ACTION removeLens_active:
IF removeLens._x AND removeLens.x = FALSE THEN
	timer.IN := FALSE;
	timer2.IN := FALSE;
	trn_removeLensDone := FALSE;
	var_process := 0;
ELSIF removeLens._x AND removeLens.x THEN
	CASE var_process OF
		0://insert parameter
			fbi_gm_removeLens.p_Init := TRUE;
			gvl_axis.fbi_motionControler.in_var_targetPosX := gvl_param.var_productInfo[gvl_param.var_currentProductID].teachPos.remove.x;
			gvl_axis.fbi_motionControler.in_var_targetPosY := gvl_param.var_productInfo[gvl_param.var_currentProductID].teachPos.remove.y;
			gvl_axis.fbi_motionControler.in_var_targetPosZ := gvl_param.var_productInfo[gvl_param.var_currentProductID].teachPos.remove.z;
			gvl_axis.fbi_motionControler.in_var_direction := eP_motionDirection.XYZ;
			IF gvl_solv.ref_ejector.input.in_flg_sensVac THEN
				var_process := 1;
			ELSE
				gvl_solv.fbi_ejector.in_var_vacMode := eP_ejeVacMode.break;
				gvl_solv.fbi_ejector.in_flg_run := TRUE;
				var_process := 20;
			END_IF
		1://move start
			gvl_axis.fbi_motionControler.in_flg_start := TRUE;
			IF gvl_axis.fbi_motionControler.out_flg_Done THEN
				var_process := 2;
			END_IF
		2://insert ejector parameter
			gvl_axis.fbi_motionControler.in_flg_start := FALSE;
			gvl_solv.fbi_ejector.in_flg_run := FALSE;
			gvl_solv.fbi_ejector.in_var_vacMode := eP_ejeVacMode.break;
			var_process := 3;
		3://break
			gvl_solv.fbi_ejector.in_flg_run := TRUE;
			IF gvl_solv.fbi_ejector.out_flg_Done THEN
				gvl_solv.fbi_ejector.in_flg_run := FALSE;
				var_process := 4;
			END_IF
		4://insert initial position
			gvl_solv.fbi_ejector.in_flg_run := FALSE;
			gvl_solv.fbi_chuck.in_var_moveMode := eP_svMoveMode.svA;
			gvl_axis.fbi_motionControler.in_var_targetPosX := gvl_param.var_productInfo[gvl_param.var_currentProductID].teachPos.initial.x;
			gvl_axis.fbi_motionControler.in_var_targetPosY := gvl_param.var_productInfo[gvl_param.var_currentProductID].teachPos.initial.y;
			gvl_axis.fbi_motionControler.in_var_targetPosZ := gvl_param.var_productInfo[gvl_param.var_currentProductID].teachPos.initial.z;
			gvl_axis.fbi_motionControler.in_var_direction := eP_motionDirection.ZYX;
			var_process := 5;
		5://move to initial position
			gvl_axis.fbi_motionControler.in_flg_start := TRUE;
			IF gvl_axis.fbi_motionControler.out_flg_Done THEN
				gvl_solv.fbi_gm_push.in_flg_run := FALSE;
				gvl_solv.fbi_gm_chuck.in_flg_run := FALSE;
				IF gvl_io.flg_fiberSens THEN
					var_process := 6;
				ELSE
					var_process := 20;
				END_IF
			END_IF
		6:
			gvl_solv.fbi_chuck.in_var_moveMode := eP_svMoveMode.svB;
			gvl_solv.fbi_push.in_var_moveMode := eP_svMoveMode.svB;
			gvl_elecylinder.fbi_axisTransport.in_var_moveMode := eP_eleMoveMode.eleB;
			gvl_solv.fbi_ejector.in_var_vacMode := eP_ejeVacMode.halt;
			gvl_axis.fbi_motionControler.in_var_targetPosX := gvl_param.var_productInfo[gvl_param.var_currentProductID].teachPos.pickUp.x;
			gvl_axis.fbi_motionControler.in_var_targetPosY := gvl_param.var_productInfo[gvl_param.var_currentProductID].teachPos.pickUp.y;
			gvl_axis.fbi_motionControler.in_var_targetPosZ := gvl_param.var_productInfo[gvl_param.var_currentProductID].teachPos.pickUp.z;
			gvl_axis.fbi_motionControler.in_var_direction := eP_motionDirection.XYZ;
			var_process := 7;
		7:
			gvl_elecylinder.fbi_axisTransport.in_flg_run := TRUE;
			gvl_solv.fbi_ejector.in_flg_run := TRUE;
			gvl_solv.fbi_chuck.in_flg_run := TRUE;
			gvl_solv.fbi_push.in_flg_run := TRUE;
			var_process := 8;
		8:
			IF gvl_io.in_wire_svChuckClose AND gvl_io.in_wire_svPushClose AND gvl_io.in_flg_eleTransportMoving THEN
				gvl_axis.fbi_motionControler.in_flg_start := TRUE;
				gvl_solv.fbi_ejector.in_flg_run := FALSE;
				gvl_elecylinder.fbi_axisTransport.in_flg_run := FALSE;
				gvl_solv.fbi_chuck.in_flg_run := FALSE;
				gvl_solv.fbi_push.in_flg_run := FALSE;
				var_process := 9;
			END_IF
		9:
			IF gvl_axis.fbi_motionControler.out_flg_Done THEN
				gvl_axis.fbi_motionControler.in_flg_start := FALSE;
				gvl_axis.fbi_motionControler.in_var_targetPosX := gvl_param.var_productInfo[gvl_param.var_currentProductID].teachPos.initial.x;
				gvl_axis.fbi_motionControler.in_var_targetPosY := gvl_param.var_productInfo[gvl_param.var_currentProductID].teachPos.initial.y;
				gvl_axis.fbi_motionControler.in_var_targetPosZ := gvl_param.var_productInfo[gvl_param.var_currentProductID].teachPos.initial.z;
				gvl_axis.fbi_motionControler.in_var_direction := eP_motionDirection.ZYX;
				var_process := 10;
			END_IF
		10:
			gvl_axis.fbi_motionControler.in_flg_start := TRUE;
			var_process := 11;
		11:
			IF gvl_axis.fbi_motionControler.out_flg_Done THEN
				gvl_axis.fbi_motionControler.in_flg_start := FALSE;
				gvl_axis.fbi_motionControler.in_var_targetPosX := gvl_param.var_productInfo[gvl_param.var_currentProductID].teachPos.remove.x;
				gvl_axis.fbi_motionControler.in_var_targetPosY := gvl_param.var_productInfo[gvl_param.var_currentProductID].teachPos.remove.y;
				gvl_axis.fbi_motionControler.in_var_targetPosZ := gvl_param.var_productInfo[gvl_param.var_currentProductID].teachPos.remove.z;
				gvl_axis.fbi_motionControler.in_var_direction := eP_motionDirection.XYZ;
				var_process := 12;
			END_IF
		12:
			gvl_axis.fbi_motionControler.in_flg_start := TRUE;
			gvl_solv.fbi_ejector.in_var_vacMode := eP_ejeVacMode.break;
			var_process := 13;
		13:
			IF gvl_axis.fbi_motionControler.out_flg_Done THEN
				gvl_solv.fbi_ejector.in_flg_run := TRUE;
				var_process := 14;	
			END_IF
		14:
			IF gvl_solv.fbi_ejector.out_flg_Done THEN
				gvl_solv.fbi_ejector.in_flg_run := FALSE;
				gvl_axis.fbi_motionControler.in_var_targetPosX := gvl_param.var_productInfo[gvl_param.var_currentProductID].teachPos.initial.x;
				gvl_axis.fbi_motionControler.in_var_targetPosY := gvl_param.var_productInfo[gvl_param.var_currentProductID].teachPos.initial.y;
				gvl_axis.fbi_motionControler.in_var_targetPosZ := gvl_param.var_productInfo[gvl_param.var_currentProductID].teachPos.initial.z;
				gvl_axis.fbi_motionControler.in_var_direction := eP_motionDirection.ZYX;
				var_process := 15;	
			END_IF
		15:
			gvl_axis.fbi_motionControler.in_flg_start := TRUE;
			gvl_solv.fbi_chuck.in_var_moveMode := eP_svMoveMode.svB;
			gvl_solv.fbi_push.in_var_moveMode := eP_svMoveMode.svB;
			gvl_elecylinder.fbi_axisTransport.in_var_moveMode := eP_eleMoveMode.eleB;
			var_process := 16;
		16:
			IF gvl_axis.fbi_motionControler.out_flg_Done THEN
				IF gvl_axis.fbi_motionControler.out_flg_Done THEN
					gvl_elecylinder.fbi_axisTransport.in_flg_run := TRUE;
					gvl_solv.fbi_chuck.in_flg_run := TRUE;
					gvl_solv.fbi_push.in_flg_run := TRUE;
					var_process := 17;
				END_IF
			END_IF
		17:
			IF gvl_io.in_wire_svChuckOpen AND gvl_io.in_wire_svPushOpen AND gvl_io.in_flg_eleTransportOrigin THEN
				gvl_elecylinder.fbi_axisTransport.in_flg_run := FALSE;
				gvl_solv.fbi_chuck.in_flg_run := FALSE;
				gvl_solv.fbi_push.in_flg_run := FALSE;
				var_process := 20;
			END_IF
		20:
			IF NOT gvl_visu.flg_btn_usingMeasurementSystem THEN
				var_process := 50;
			ELSE
				fbi_gm_removeLens.p_Init := TRUE;
				fbi_gm_removeLens.in_flg_run := FALSE;
				var_process := 21;
			END_IF
		21:
			fbi_gm_removeLens.p_Init := FALSE;
			fbi_gm_removeLens.in_flg_run := TRUE;
			var_process := 22;
		22:
			fbi_gm_removeLens.in_flg_run := FALSE;
			IF fbi_gm_removeLens.out_flg_Done THEN
				var_process := 50;
			END_IF
			
		50:
			gvl_solv.fbi_ejector.in_flg_run := FALSE;
			trn_removeLensDone := TRUE;
	END_CASE
	fbi_gm_removeLens(in_flg_run:= , out_flg_Done=> );
	timer(IN:= , PT:= T#0.5S , Q=> , ET=> );
	timer2(IN:= , PT:= T#0.5S , Q=> , ET=> );
END_IF
END_ACTION

END_FUNCTION_BLOCK

// ---- FBs/fb_lensTranport.TcPOU
FUNCTION_BLOCK fb_lensTranport
VAR_INPUT
END_VAR
VAR_OUTPUT
END_VAR
VAR
	SFCInit: bool;
	trn_wattingForLensDone: BOOL;
	trn_connectionCheckDone: BOOL;
	flg_buf_gateLengthISSuccessed: BOOL;
	flg_buf_dummySignal: BOOL;
	trn_chuckDone: BOOL;
	var_chuckCount: INT;
	trn_transportDone: BOOL;
	trn_waitTakingLensDone: BOOL;
	trn_moveToHomeDone: BOOL;
	fbi_getCav: fb_getCav;
	trn_readCavDone: BOOL;
	trn_gm_chuckDone: BOOL;
	trn_gm_transportDone: BOOL;
	trn_gm_moveToHomeDone: BOOL;
	trn_cavCheckDone: BOOL;
	fbi_delayTimer: TON;
	trn_AddCountDone: BOOL;
	var_process: INT;
	flg_chuckDone: BOOL;
	flg_pushDone: BOOL;
	trn_LensCheckDone: BOOL;
END_VAR

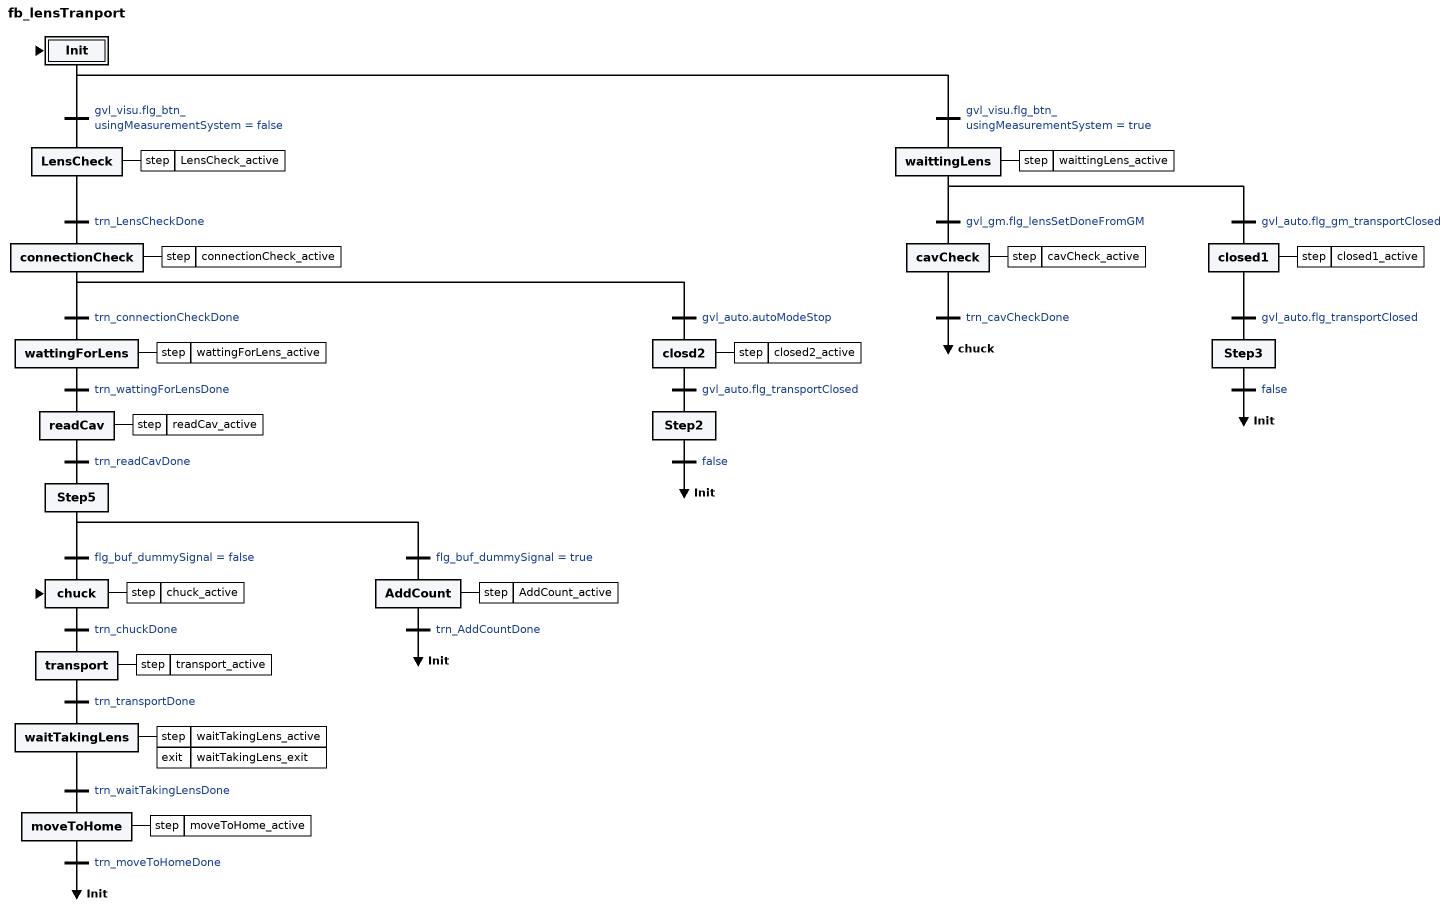
INITIAL_STEP Init:
END_STEP
TRANSITION FROM Init TO LensCheck
    := gvl_visu.flg_btn_usingMeasurementSystem = false;
END_TRANSITION
TRANSITION FROM Init TO waittingLens
    := gvl_visu.flg_btn_usingMeasurementSystem = true;
END_TRANSITION
STEP waittingLens:
    waittingLens_active(N);  // step action
END_STEP
TRANSITION FROM waittingLens TO cavCheck
    := gvl_gm.flg_lensSetDoneFromGM;
END_TRANSITION
STEP cavCheck:
    cavCheck_active(N);  // step action
END_STEP
TRANSITION FROM cavCheck TO chuck
    := trn_cavCheckDone;
END_TRANSITION
TRANSITION FROM waittingLens TO closed1
    := gvl_auto.flg_gm_transportClosed;
END_TRANSITION
STEP closed1:
    closed1_active(N);  // step action
END_STEP
TRANSITION FROM closed1 TO Step3
    := gvl_auto.flg_transportClosed;
END_TRANSITION
STEP Step3:
END_STEP
TRANSITION FROM Step3 TO Init
    := false;
END_TRANSITION
STEP LensCheck:
    LensCheck_active(N);  // step action
END_STEP
TRANSITION FROM LensCheck TO connectionCheck
    := trn_LensCheckDone;
END_TRANSITION
STEP connectionCheck:
    connectionCheck_active(N);  // step action
END_STEP
TRANSITION FROM connectionCheck TO wattingForLens
    := trn_connectionCheckDone;
END_TRANSITION
STEP wattingForLens:
    wattingForLens_active(N);  // step action
END_STEP
TRANSITION FROM wattingForLens TO readCav
    := trn_wattingForLensDone;
END_TRANSITION
TRANSITION FROM connectionCheck TO closd2
    := gvl_auto.autoModeStop;
END_TRANSITION
STEP closd2:
    closed2_active(N);  // step action
END_STEP
TRANSITION FROM closd2 TO Step2
    := gvl_auto.flg_transportClosed;
END_TRANSITION
STEP Step2:
END_STEP
TRANSITION FROM Step2 TO Init
    := false;
END_TRANSITION
STEP readCav:
    readCav_active(N);  // step action
END_STEP
TRANSITION FROM readCav TO Step5
    := trn_readCavDone;
END_TRANSITION
STEP Step5:
END_STEP
TRANSITION FROM Step5 TO chuck
    := flg_buf_dummySignal = false;
END_TRANSITION
TRANSITION FROM Step5 TO AddCount
    := flg_buf_dummySignal = true;
END_TRANSITION
STEP AddCount:
    AddCount_active(N);  // step action
END_STEP
TRANSITION FROM AddCount TO Init
    := trn_AddCountDone;
END_TRANSITION
STEP chuck:
    chuck_active(N);  // step action
END_STEP
TRANSITION FROM chuck TO transport
    := trn_chuckDone;
END_TRANSITION
STEP transport:
    transport_active(N);  // step action
END_STEP
TRANSITION FROM transport TO waitTakingLens
    := trn_transportDone;
END_TRANSITION
STEP waitTakingLens:
    waitTakingLens_active(N);  // step action
    waitTakingLens_exit(P0);  // exit action
END_STEP
TRANSITION FROM waitTakingLens TO moveToHome
    := trn_waitTakingLensDone;
END_TRANSITION
STEP moveToHome:
    moveToHome_active(N);  // step action
END_STEP
TRANSITION FROM moveToHome TO Init
    := trn_moveToHomeDone;
END_TRANSITION

ACTION AddCount_active:
IF AddCount._x AND AddCount.x = FALSE THEN
	trn_AddCountDone := FALSE;
ELSIF AddCount._x AND AddCount.x THEN
	trn_AddCountDone := TRUE;
END_IF
END_ACTION

ACTION cavCheck_active:
IF cavCheck._x AND cavCheck.x = FALSE THEN
	trn_cavCheckDone := FALSE;
ELSIF cavCheck._x AND cavCheck.x THEN
	gvl_auto.cavNo := gvl_gm.var_buf_tranportCav;
	gvl_auto.flg_buf_gateLengthIsPassed := gvl_gm.flg_buf_gateLengthIsPassed;
	trn_cavCheckDone := TRUE;
END_IF
END_ACTION

ACTION chuck_active:
IF chuck._x AND chuck.x = FALSE THEN
	gvl_gm.flg_lensRequest := FALSE;
	trn_chuckDone := FALSE;
	gvl_auto.flg_gateData_Tx := FALSE;
	gvl_solv.fbi_chuck.in_flg_run := FALSE;
	gvl_solv.fbi_push.in_flg_run := FALSE;
	var_chuckCount := -11;
ELSIF chuck._x AND chuck.x THEN
	CASE var_chuckCount OF
		-11:
			IF gvl_param.var_productInfo[gvl_param.var_currentProductID].flg_mode_stocker THEN
				var_chuckCount := -10; // Mode 1
			ELSE
				var_chuckCount := 0;  // Mode 0
			END_IF
		
		// Mode 1: 押す →　解除　→ チャック →　押す
		-10:
			gvl_solv.fbi_push.in_var_moveMode := eP_svMoveMode.svB;
			gvl_solv.fbi_push.in_flg_run := TRUE;
			var_chuckCount := -9;
		-9://close
			IF gvl_solv.fbi_push.out_flg_Done THEN
				gvl_solv.fbi_push.in_flg_run := FALSE;
				var_chuckCount := -8;
			END_IF
		-8:		
			gvl_solv.fbi_push.in_var_moveMode := eP_svMoveMode.svA;
			gvl_solv.fbi_push.in_flg_run := TRUE;
			var_chuckCount := -7;
		-7://open
			IF gvl_solv.fbi_push.out_flg_Done THEN
				gvl_solv.fbi_push.in_flg_run := FALSE;
				var_chuckCount := -6;
			END_IF
		-6:
			gvl_solv.fbi_chuck.in_var_moveMode := eP_svMoveMode.svB;
			gvl_solv.fbi_chuck.in_flg_run := TRUE;
			var_chuckCount := -5;
		-5://push close
			IF gvl_solv.fbi_chuck.out_flg_Done THEN
				gvl_solv.fbi_chuck.in_flg_run := FALSE;
				var_chuckCount := -4;
			END_IF
		-4:
			gvl_solv.fbi_push.in_var_moveMode := eP_svMoveMode.svB;
			gvl_solv.fbi_push.in_flg_run := TRUE;
			var_chuckCount := -3;
		-3://close
			
			IF gvl_solv.fbi_push.out_flg_Done THEN
				gvl_solv.fbi_push.in_flg_run := FALSE;
				var_chuckCount := 12;
			END_IF
		
		// Mode 0: チャック → 解除 → 押す → チャック
		0:
			gvl_solv.fbi_chuck.in_var_moveMode := eP_svMoveMode.svB;
			gvl_solv.fbi_chuck.in_flg_run := TRUE;
			var_chuckCount := 1;
		1://close
			
			IF gvl_solv.fbi_chuck.out_flg_Done THEN
				gvl_solv.fbi_chuck.in_flg_run := FALSE;
				var_chuckCount := 2;
			END_IF
		2:		
			gvl_solv.fbi_chuck.in_var_moveMode := eP_svMoveMode.svA;
			gvl_solv.fbi_chuck.in_flg_run := TRUE;
			var_chuckCount := 3;
		3://open
			
			IF gvl_solv.fbi_chuck.out_flg_Done THEN
				var_chuckCount := 4;
			END_IF
		4:
			gvl_solv.fbi_push.in_var_moveMode := eP_svMoveMode.svB;
			gvl_solv.fbi_push.in_flg_run := TRUE;
			var_chuckCount := 5;
		5://push close
			
			IF gvl_solv.fbi_push.out_flg_Done THEN
				gvl_solv.fbi_push.in_flg_run := FALSE;
				gvl_solv.fbi_chuck.in_flg_run := FALSE;
				var_chuckCount := 6;
			END_IF
		6:
			
			gvl_solv.fbi_chuck.in_var_moveMode := eP_svMoveMode.svB;
			gvl_solv.fbi_chuck.in_flg_run := TRUE;
			var_chuckCount := 7;
		7://close
			
			IF gvl_solv.fbi_chuck.out_flg_Done THEN
				gvl_solv.fbi_chuck.in_flg_run := FALSE;
				var_chuckCount := 12;
			END_IF
		8:
			
			gvl_solv.fbi_chuck.in_var_moveMode := eP_svMoveMode.svA;
			gvl_solv.fbi_chuck.in_flg_run := TRUE;
			var_chuckCount := 9;
		9://open
			
			IF gvl_solv.fbi_chuck.out_flg_Done THEN
				gvl_solv.fbi_chuck.in_flg_run := FALSE;
				var_chuckCount := 10;
			END_IF
		10:
			
			gvl_solv.fbi_chuck.in_var_moveMode := eP_svMoveMode.svB;
			gvl_solv.fbi_chuck.in_flg_run := TRUE;
			var_chuckCount := 11;
		11://close
			
			IF gvl_solv.fbi_chuck.out_flg_Done THEN
				var_chuckCount := 12;
			END_IF
		12://gate measurement
			IF gvl_visu.flg_btn_gateMeasurementIsNone THEN
				IF flg_buf_gateLengthISSuccessed THEN
					gvl_auto.gateLengthIsPassed := TRUE;
				ELSIF gvl_auto.flg_buf_gateLengthIsPassed THEN
					gvl_auto.gateLengthIsPassed := TRUE;
				ELSE
					gvl_auto.gateLengthIsPassed := FALSE;
				END_IF
			ELSE
				IF gvl_io.var_gateLength > gvl_param.var_productInfo[gvl_param.var_currentProductID].gateLength_max OR gvl_io.var_gateLength < gvl_param.var_productInfo[gvl_param.var_currentProductID].gateLength_min THEN
					gvl_auto.gateLengthIsPassed := FALSE;
				ELSE
					gvl_auto.gateLengthIsPassed := TRUE;
				END_IF
				gvl_auto.flg_gateData_Tx := TRUE;
				
			END_IF
			var_chuckCount := 13;
		13:
			gvl_solv.fbi_chuck.in_flg_run := FALSE;
			gvl_elecylinder.fbi_axisRotary.in_flg_run := FALSE;
			gvl_elecylinder.fbi_axisRotary.in_var_moveMode := eP_eleMoveMode.eleB;
			IF gvl_visu.flg_btn_RotaryIsNotUse THEN
				var_chuckCount := 16;
			ELSE
				var_chuckCount := 14;
			END_IF
		14:
			gvl_elecylinder.fbi_axisRotary.in_flg_run := TRUE;
			var_chuckCount := 15;
		15:
			IF gvl_elecylinder.fbi_axisRotary.out_flg_Done THEN
				gvl_elecylinder.fbi_axisRotary.in_flg_run := FALSE;
				var_chuckCount := 16;
			END_IF
		16:
			trn_chuckDone := TRUE;
	END_CASE
END_IF
END_ACTION

ACTION closed1_active:
IF closed1._x AND closed1.x = FALSE THEN
	gvl_auto.flg_transportClosed := FALSE;
	gvl_elecylinder.fbi_axisTransport.in_flg_run := FALSE;
	gvl_elecylinder.fbi_axisRotary.in_flg_run:= FALSE;
	gvl_elecylinder.fbi_axisTransport.in_var_moveMode := eP_eleMoveMode.eleB;
	gvl_elecylinder.fbi_axisRotary.in_var_moveMode:= eP_eleMoveMode.eleB;
	var_process := 0;
ELSIF closed1._x AND closed1.x THEN
	CASE var_process OF
		0:
			gvl_elecylinder.fbi_axisRotary.in_flg_run:= TRUE;
			var_process := 1;
		1:
			IF gvl_elecylinder.fbi_axisRotary.out_flg_Done THEN
				gvl_elecylinder.fbi_axisRotary.in_flg_run:= FALSE;
				var_process := 2;
			END_IF
		2:
			gvl_elecylinder.fbi_axisTransport.in_flg_run := TRUE;
			var_process := 3;
		3:
			IF gvl_elecylinder.fbi_axisTransport.out_flg_Done THEN
				gvl_elecylinder.fbi_axisTransport.in_flg_run:= FALSE;
				gvl_auto.flg_transportClosed := TRUE;
			END_IF
	END_CASE
END_IF
END_ACTION

ACTION closed2_active:
IF closd2._x AND closd2.x = FALSE THEN
	gvl_auto.flg_transportClosed := FALSE;
ELSIF closd2._x AND closd2.x THEN
	gvl_io.flg_requestLens := FALSE;
	gvl_auto.flg_transportClosed := true;
END_IF
END_ACTION

ACTION connectionCheck_active:
IF connectionCheck._x AND connectionCheck.x = FALSE THEN
	trn_connectionCheckDone:= FALSE;
	gvl_io.flg_requestLens := TRUE;
ELSIF connectionCheck._x AND connectionCheck.x THEN
	IF gvl_io.in_bitNumber0 
		AND gvl_io.in_bitNumber1
		AND gvl_io.in_bitNumber2
		AND gvl_io.in_bitNumber3 OR gvl_debug.cavConecctSkip THEN
		trn_connectionCheckDone:= TRUE;
	END_IF
	IF NOT gvl_visu.flg_btn_vacSensOn THEN
		gvl_error.flg_fiberSens := gvl_io.flg_fiberSens;
	END_IF
END_IF
END_ACTION

ACTION LensCheck_active:
IF LensCheck._x AND LensCheck.x = FALSE THEN
	trn_LensCheckDone := FALSE;
ELSIF LensCheck._x AND LensCheck.x THEN
	IF NOT gvl_visu.flg_btn_vacSensOn THEN
		IF gvl_io.flg_fiberSens OR gvl_debug.out_fiberSens THEN
			gvl_error.flg_fiberSens := TRUE;	
		ELSE
			trn_LensCheckDone := TRUE;
		END_IF
	ELSE
		trn_LensCheckDone := TRUE;
	END_IF
END_IF
END_ACTION

ACTION moveToHome_active:
IF moveToHome._x AND moveToHome.x = FALSE THEN
	trn_moveToHomeDone := FALSE;
	gvl_elecylinder.fbi_axisTransport.in_flg_run := FALSE;
	gvl_elecylinder.fbi_axisTransport.in_var_moveMode := eP_eleMoveMode.eleA;
	gvl_elecylinder.fbi_axisRotary.in_var_moveMode := eP_eleMoveMode.eleA;
	var_process := 0;
ELSIF moveToHome._x AND moveToHome.x THEN
	CASE var_process OF
		0:
			gvl_elecylinder.fbi_axisTransport.in_flg_run := TRUE;
			var_process := 1;
		1:
			IF gvl_elecylinder.fbi_axisTransport.out_flg_Done THEN
				gvl_elecylinder.fbi_axisTransport.in_flg_run := FALSE;
				var_process := 2;
			END_IF
		2:
			gvl_elecylinder.fbi_axisRotary.in_flg_run := TRUE;
			var_process := 3;
		3:
			IF gvl_elecylinder.fbi_axisRotary.out_flg_Done THEN
				gvl_elecylinder.fbi_axisRotary.in_flg_run := FALSE;
				var_process := 4;
			END_IF
		4:
			IF gvl_elecylinder.ref_axis_transport.input.in_flg_sensA AND gvl_elecylinder.ref_axis_rotary.input.in_flg_sensA THEN
				trn_moveToHomeDone := TRUE;
			END_IF
	END_CASE
	
	
	//
END_IF
END_ACTION

PROPERTY p_Init : bool
GET
p_init := THIS^.SFCInit;
END_GET
SET
THIS^.SFCInit := p_init;
END_SET
END_PROPERTY

ACTION readCav_active:
IF readCav._x AND readCav.x = FALSE THEN
	trn_readCavDone := FALSE;
	THIS^.fbi_getCav();
	fbi_getCav.in_flg_run := FALSE;
	fbi_delayTimer.IN := FALSE;
ELSIF readCav._x AND readCav.x THEN
	THIS^.fbi_getCav();
	fbi_delayTimer.IN := TRUE;
	THIS^.fbi_getCav.in_flg_run := fbi_delayTimer.Q;
	IF THIS^.fbi_getCav.out_flg_Done THEN
		IF gvl_debug.flg_debug_run THEN
			gvl_auto.cavNo := gvl_debug.var_cav;
		ELSE
			gvl_auto.cavNo := THIS^.fbi_getCav.out_var_cav;
		END_IF
		trn_readCavDone := TRUE;
	ELSIF THIS^.fbi_getCav.out_flg_error THEN
		IF gvl_debug.flg_debug_run THEN
			gvl_auto.cavNo := gvl_debug.var_cav;
		ELSE
			gvl_auto.cavNo := 0;
		END_IF
		trn_readCavDone := TRUE;
	END_IF
END_IF

fbi_delayTimer(IN:= , PT:=T#200MS , Q=> , ET=> );
END_ACTION

ACTION transport_active:
IF transport._x AND transport.x = FALSE THEN
	gvl_elecylinder.fbi_axisTransport.in_flg_run := FALSE;
	trn_transportDone := FALSE;
	gvl_elecylinder.fbi_axisTransport.in_var_moveMode := eP_eleMoveMode.eleB;
	var_process := 0;
ELSIF transport._x AND transport.x THEN
	CASE var_process OF
		0:
			IF NOT gvl_auto.flg_sampling THEN
				gvl_elecylinder.fbi_axisTransport.in_flg_run := TRUE;
				var_process := 1;
			END_IF
		1:
			IF gvl_elecylinder.fbi_axisTransport.out_flg_Done THEN
				gvl_elecylinder.fbi_axisTransport.in_flg_run := FALSE;
				trn_transportDone := TRUE;
			END_IF
	END_CASE
END_IF
END_ACTION

ACTION waitTakingLens_active:
IF waitTakingLens._x AND waitTakingLens.x = FALSE THEN
	trn_waitTakingLensDone := FALSE;
	flg_chuckDone:= FALSE;
	flg_pushDone := FALSE;
	gvl_solv.fbi_chuck.in_var_moveMode := eP_svMoveMode.svA;
	gvl_solv.fbi_push.in_var_moveMode := eP_svMoveMode.svA;
	gvl_auto.buf_cavNo := gvl_auto.cavNo;
	gvl_auto.flg_gateLength := gvl_auto.gateLengthIsPassed;
ELSIF waitTakingLens._x AND waitTakingLens.x THEN
	gvl_auto.requirementToPickUpLens := TRUE;
	IF gvl_auto.lensVacuumDone THEN
		gvl_auto.buf_gateLength := gvl_visu.var_gateLengthList[0];
		gvl_solv.fbi_chuck.in_flg_run := TRUE;
		gvl_solv.fbi_push.in_flg_run := TRUE;
	END_IF
	IF gvl_solv.fbi_chuck.out_flg_Done THEN
		flg_chuckDone := TRUE;
	END_IF
	IF gvl_solv.fbi_push.out_flg_Done THEN
		flg_pushDone := TRUE;
	END_IF
	IF flg_chuckDone AND flg_pushDone THEN
		gvl_solv.fbi_chuck.in_flg_run := FALSE;
		gvl_solv.fbi_push.in_flg_run := FALSE;
		gvl_auto.chuckopenDone := TRUE;
	END_IF
	IF gvl_auto.pickUpLnesDone THEN
		trn_waitTakingLensDone := TRUE;
	END_IF
END_IF
END_ACTION

ACTION waitTakingLens_exit:
gvl_auto.lensVacuumDone := FALSE;
gvl_auto.requirementToPickUpLens := FALSE;
gvl_auto.chuckopenDone := FALSE;
gvl_auto.pickUpLnesDone := FALSE;
END_ACTION

ACTION waittingLens_active:
IF waittingLens._x AND waittingLens.x = FALSE THEN
	gvl_gm.flg_lensRequest := FALSE;
	gvl_gm.flg_lensSetDoneFromGM := FALSE;
	IF NOT gvl_visu.flg_btn_vacSensOn THEN
		gvl_error.flg_fiberSens := gvl_io.flg_fiberSens;
	END_IF
ELSIF waittingLens._x AND waittingLens.x THEN
	gvl_gm.flg_lensRequest := TRUE;
END_IF
END_ACTION

ACTION wattingForLens_active:
IF wattingForLens._x AND wattingForLens.x = FALSE THEN
	trn_wattingForLensDone := FALSE;
	flg_buf_gateLengthISSuccessed := FALSE;
	flg_buf_dummySignal := FALSE;
ELSIF wattingForLens._x AND wattingForLens.x THEN
	//gate
	IF gvl_IO.flg_gateLengthIsSuccessed OR gvl_debug.flg_passingMeasurement THEN
		flg_buf_gateLengthISSuccessed := TRUE;
	END_IF
	//dummy signal
	IF gvl_io.flg_dummySiganl THEN
		flg_buf_dummySignal := TRUE;
	END_IF
	//lens set done
	IF NOT gvl_visu.flg_btn_vacSensOn THEN
		IF gvl_io.flg_lensSetDone AND gvl_io.flg_fiberSens OR gvl_debug.out_lensSetDone THEN
			gvl_io.flg_requestLens := FALSE;
			trn_wattingForLensDone := TRUE;
		ELSIF gvl_io.flg_lensSetDone AND gvl_io.flg_fiberSens = FALSE THEN
			gvl_error.flg_fiberSens := TRUE;
		END_IF
	ELSE
		IF gvl_io.flg_lensSetDone OR gvl_debug.out_lensSetDone  THEN
			gvl_io.flg_requestLens := FALSE;
			trn_wattingForLensDone := TRUE;
		END_IF
	END_IF
END_IF
END_ACTION

END_FUNCTION_BLOCK

// ---- FBs/fb_getCav.TcPOU
FUNCTION_BLOCK fb_getCav
VAR_INPUT
	in_flg_run: BOOL;
END_VAR
VAR_OUTPUT
	out_flg_run: BOOL;
	out_flg_Done: BOOL;
	out_flg_error: BOOL;
	out_var_cav: INT;
END_VAR
VAR
	var_iCav : INT;
	fbi_r_trig: R_TRIG;
	var_process: INT;
END_VAR

out_flg_run := in_flg_run;
fbi_r_trig(CLK:=in_flg_run , Q=> );
IF fbi_r_trig.Q THEN
	var_process := 1;
END_IF
CASE var_process OF
	0:
			
	1:
		var_iCav.0 := gvl_io.flg_bitNumber0;
		var_iCav.1 := gvl_io.flg_bitNumber1;
		var_iCav.2 := gvl_io.flg_bitNumber2;
		var_iCav.3 := gvl_io.flg_bitNumber3;
		out_var_cav := var_iCav;
		var_process := 2;
	2:
		IF out_var_cav > gvl_param.var_productInfo[gvl_param.var_currentProductID].cavQty  OR out_var_cav = 0 THEN
			out_flg_error := TRUE;
			var_process := 4;
		ELSE
			var_process := 3;
		END_IF
	3:
		out_flg_Done := TRUE;
		var_process := 4;
	4:
		out_flg_error := FALSE;
		out_flg_Done := FALSE;
		var_process := 0;
END_CASE

END_FUNCTION_BLOCK

// ---- FBs/fb_palletizeing.TcPOU
FUNCTION_BLOCK fb_palletizeing
VAR_INPUT
END_VAR
VAR_OUTPUT
END_VAR
VAR
	SFCInit: BOOL;
	fbi_coordinateCal: fb_coordinateCal;
	fbi_exchangeTraySystem: fb_exchangeTraySystem;
	trn_pickUpLensDone: BOOL;
	trn_forTray: BOOL;
	trn_forGarbage: BOOL;
	trn_forSample: BOOL;
	trn_trayDone: BOOL;
	trn_garbageDone: BOOL;
	trn_sampleDone: BOOL;
	trn_calculateDone: BOOL;
	var_targetPosX: LREAL;
	var_targetPosY: LREAL;
	var_targetPosZ: LREAL;
	var_process: INT;
	flg_trayIsFull: BOOL;
	flg_sampleIsBusy: BOOL;
	flg_trayIsNotFull: BOOL;
	flg_sampleCavCheck: ARRAY[1..8] OF BOOL;
	var_i: INT;
	flg_bufCavChcek: BOOL;
	trn_moveToInitPosDone: BOOL;
	trn_notTrayChange: BOOL;
	trn_trayChange: BOOL;
	flg_pocketIsNotFull: BOOL;
	trn_trayChangeDone			: BOOL;
	var_cav						: INT;
	trn_DataSamplingDone		: BOOL;
	fbi_vacuumRetry				: fb_vacuumRetry;
	vacuumRetryTimer			: TON;
	var_i_clear					: INT;
	flg_allLensIsNotSet			: BOOL;
	flg_axisSample_Done			: BOOL;
	flg_axisXY_move_Sample_Done	: BOOL;
	fb_TON_delay				: TON;
	fb_TON_delay_error			: TON;
	flg_sample_need				: BOOL;
END_VAR

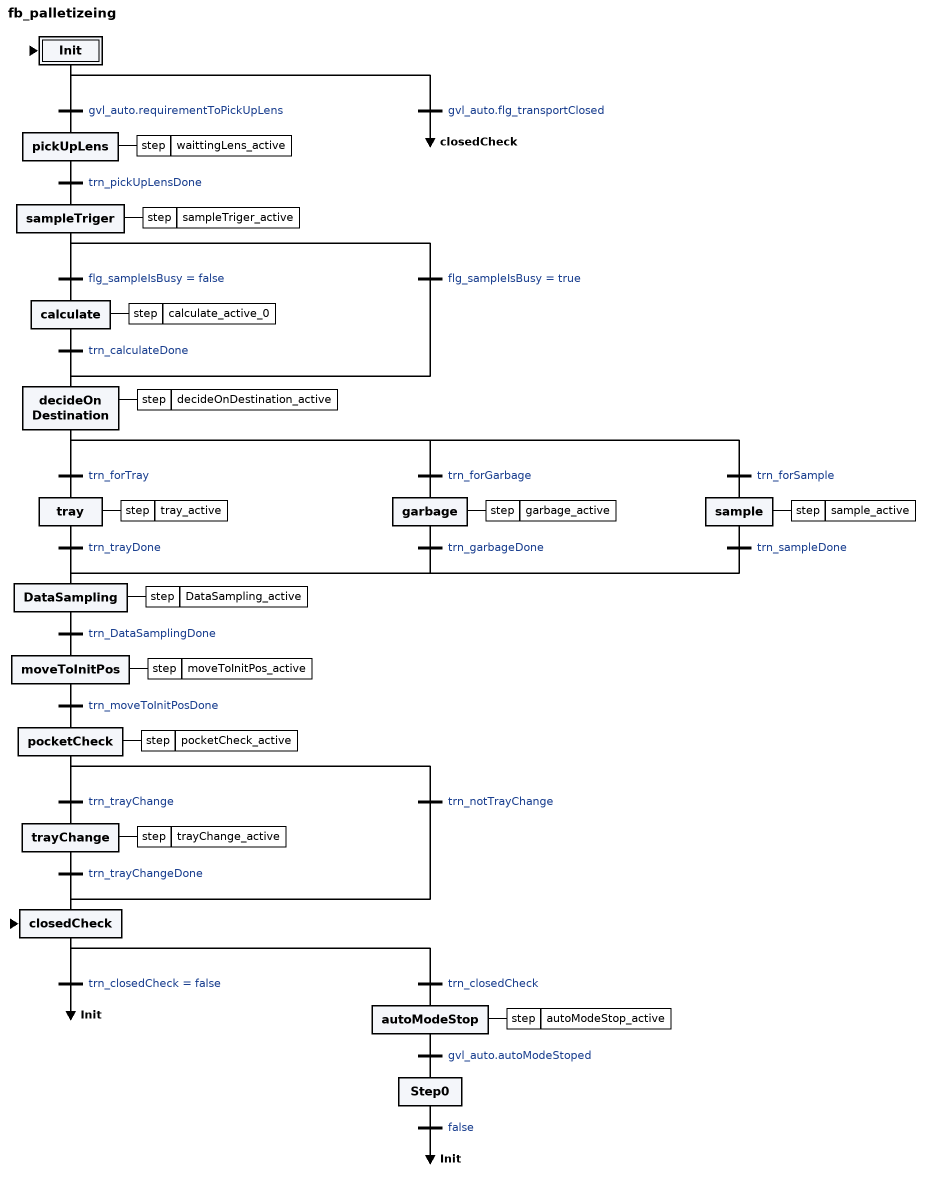
INITIAL_STEP Init:
END_STEP
TRANSITION FROM Init TO pickUpLens
    := gvl_auto.requirementToPickUpLens;
END_TRANSITION
TRANSITION FROM Init TO closedCheck
    := gvl_auto.flg_transportClosed;
END_TRANSITION
STEP pickUpLens:
    waittingLens_active(N);  // step action
END_STEP
TRANSITION FROM pickUpLens TO sampleTriger
    := trn_pickUpLensDone;
END_TRANSITION
STEP sampleTriger:
    sampleTriger_active(N);  // step action
END_STEP
TRANSITION FROM sampleTriger TO calculate
    := flg_sampleIsBusy = false;
END_TRANSITION
STEP calculate:
    calculate_active_0(N);  // step action
END_STEP
TRANSITION FROM calculate TO decideOnDestination
    := trn_calculateDone;
END_TRANSITION
TRANSITION FROM sampleTriger TO decideOnDestination
    := flg_sampleIsBusy = true;
END_TRANSITION
STEP decideOnDestination:
    decideOnDestination_active(N);  // step action
END_STEP
TRANSITION FROM decideOnDestination TO tray
    := trn_forTray;
END_TRANSITION
STEP tray:
    tray_active(N);  // step action
END_STEP
TRANSITION FROM tray TO DataSampling
    := trn_trayDone;
END_TRANSITION
TRANSITION FROM decideOnDestination TO garbage
    := trn_forGarbage;
END_TRANSITION
STEP garbage:
    garbage_active(N);  // step action
END_STEP
TRANSITION FROM garbage TO DataSampling
    := trn_garbageDone;
END_TRANSITION
TRANSITION FROM decideOnDestination TO sample
    := trn_forSample;
END_TRANSITION
STEP sample:
    sample_active(N);  // step action
END_STEP
TRANSITION FROM sample TO DataSampling
    := trn_sampleDone;
END_TRANSITION
STEP DataSampling:
    DataSampling_active(N);  // step action
END_STEP
TRANSITION FROM DataSampling TO moveToInitPos
    := trn_DataSamplingDone;
END_TRANSITION
STEP moveToInitPos:
    moveToInitPos_active(N);  // step action
END_STEP
TRANSITION FROM moveToInitPos TO pocketCheck
    := trn_moveToInitPosDone;
END_TRANSITION
STEP pocketCheck:
    pocketCheck_active(N);  // step action
END_STEP
TRANSITION FROM pocketCheck TO trayChange
    := trn_trayChange;
END_TRANSITION
STEP trayChange:
    trayChange_active(N);  // step action
END_STEP
TRANSITION FROM trayChange TO closedCheck
    := trn_trayChangeDone;
END_TRANSITION
TRANSITION FROM pocketCheck TO closedCheck
    := trn_notTrayChange;
END_TRANSITION
STEP closedCheck:
END_STEP
TRANSITION FROM closedCheck TO Init
    := trn_closedCheck = false;
END_TRANSITION
TRANSITION FROM closedCheck TO autoModeStop
    := trn_closedCheck;
END_TRANSITION
STEP autoModeStop:
    autoModeStop_active(N);  // step action
END_STEP
TRANSITION FROM autoModeStop TO Step0
    := gvl_auto.autoModeStoped;
END_TRANSITION
STEP Step0:
END_STEP
TRANSITION FROM Step0 TO Init
    := false;
END_TRANSITION

ACTION autoModeStop_active:
IF autoModeStop._x AND autoModeStop.x = FALSE THEN
	gvl_auto.autoModeStoped := FALSE;
ELSIF autoModeStop._x AND autoModeStop.x THEN
	gvl_auto.autoModeStoped := TRUE;
END_IF
END_ACTION

ACTION calculate_active_0:
IF calculate._x AND calculate.x = FALSE THEN
	var_process := 0;
	fbi_coordinateCal.in_flg_run := FALSE;
	trn_calculateDone := FALSE;
	flg_trayIsNotFull := FALSE;
ELSIF calculate._x AND calculate.x THEN
	CASE var_process OF
		0:
			var_process := 1;
		1:
			IF  gvl_auto.buf_cavNo <> 0 THEN
				IF  gvl_auto.pocketNo[gvl_auto.buf_cavNo] < gvl_param.var_productInfo[gvl_param.var_currentProductID].pocketSumQty  THEN
					flg_trayIsNotFull := TRUE;
				END_IF
				var_process := 2;
			ELSE
				var_process := 3;
			END_IF
		2:
			fbi_coordinateCal.in_flg_run := TRUE;
			IF fbi_coordinateCal.out_flg_Done THEN
				fbi_coordinateCal.in_flg_run := FALSE;
				var_process := 3;
			END_IF
		3:
			trn_calculateDone := TRUE;
			
	END_CASE
END_IF
fbi_coordinateCal(
	in_flg_run:= , 
	out_flg_run=> , 
	var_ref_productInfo:= gvl_param.var_productInfo[gvl_param.var_currentProductID], 
	in_var_cavNo:= gvl_auto.buf_cavNo, 
	in_var_pocketNo:= gvl_auto.pocketNo[gvl_auto.buf_cavNo] + 1, 
	in_var_calculateMode:= eP_calculateMode.Affine, 
	out_flg_busy=> , 
	out_flg_Done=> , 
	out_var_X=> var_targetPosX, 
	out_var_Y=> var_targetPosY, 
	out_var_Z=> var_targetPosZ);
END_ACTION

ACTION DataSampling_active:
IF DataSampling._x AND DataSampling.x = FALSE THEN
	gvl_auto.flg_dataSampling_run := FALSE;
	trn_DataSamplingDone := FALSE;
ELSIF DataSampling._x AND DataSampling.x THEN
	gvl_auto.flg_dataSampling_run := TRUE;
	trn_DataSamplingDone := TRUE;
END_IF
END_ACTION

ACTION decideOnDestination_active:
IF decideOnDestination._x AND decideOnDestination.x = FALSE THEN
	trn_forTray := FALSE;
	trn_forGarbage := FALSE;
	trn_forSample := FALSE;
	gvl_auto.flg_DataSample_nonDefective := FALSE;
	gvl_auto.flg_DataSample_defective := FALSE;
	gvl_auto.flg_DataSamle_sample := FALSE;
	IF gvl_auto.flg_pocketCountCheck THEN
		gvl_auto.pocketNo[gvl_auto.flg_pocketCountCheck_cav] := gvl_auto.pocketNo[gvl_auto.flg_pocketCountCheck_cav] -1;
	END_IF
ELSIF decideOnDestination._x AND decideOnDestination.x THEN
	gvl_auto.flg_pocketCountCheck_cav := gvl_auto.buf_cavNo;
	gvl_auto.flg_axisIsPcikingUp := FALSE;
	IF flg_trayIsNotFull AND gvl_auto.flg_gateLength AND gvl_auto.buf_cavNo <> 0 AND NOT flg_sampleIsBusy THEN
	//tray
		gvl_auto.flg_pocketCountCheck := TRUE;
		trn_forTray := TRUE;
		gvl_auto.flg_DataSample_nonDefective := TRUE;
	ELSIF flg_sampleIsBusy AND flg_sample_need THEN
	//sample
		gvl_auto.flg_pocketCountCheck := TRUE;
		trn_forSample := TRUE;
		gvl_auto.flg_DataSamle_sample := TRUE;
	ELSE
	//garbage
		IF NOT gvl_auto.flg_gm_eleIsDown THEN
			trn_forGarbage := TRUE;
			gvl_auto.flg_DataSample_defective := TRUE;
		END_IF
	END_IF
END_IF
END_ACTION

ACTION garbage_active:
IF garbage._x AND garbage.x = FALSE THEN
	gvl_axis.fbi_motionControler.in_flg_start := FALSE;
	gvl_solv.fbi_ejector.in_flg_run := FALSE;
	trn_garbageDone := FALSE;
	var_process := 0;
	gvl_auto.var_defectiveLens[gvl_auto.buf_cavNo] := gvl_auto.var_defectiveLens[gvl_auto.buf_cavNo] + 1;
ELSIF garbage._x AND garbage.x THEN
	CASE var_process OF
//		-2:
//			gvl_elecylinder.fbi_axisSample.in_flg_run := FALSE;
//			gvl_elecylinder.fbi_axisSample.in_var_moveMode := eP_eleMoveMode.eleA;
//			gvl_axis.fbi_motionControler.in_flg_start := FALSE;
//			IF gvl_io.flg_frontSaftyDoor THEN
//				gvl_elecylinder.fbi_axisSample.in_flg_run := TRUE;
//				var_process := -1;
//			END_IF
//		-1:
//			IF gvl_elecylinder.fbi_axisSample.out_flg_Done THEN
//				gvl_elecylinder.fbi_axisSample.in_flg_run := FALSE;
//				var_process := 0;
//			END_IF
		0:
			gvl_axis.fbi_motionControler.in_var_targetPosX := gvl_param.var_productInfo[gvl_param.var_currentProductID].teachPos.remove.x;
			gvl_axis.fbi_motionControler.in_var_targetPosY := gvl_param.var_productInfo[gvl_param.var_currentProductID].teachPos.remove.y;
			gvl_axis.fbi_motionControler.in_var_targetPosZ := gvl_param.var_productInfo[gvl_param.var_currentProductID].teachPos.remove.z;
			gvl_axis.fbi_motionControler.in_var_direction := eP_motionDirection.Y_X_Z;
			var_process := 1;
		1:
			gvl_axis.fbi_motionControler.in_flg_start := TRUE;
			var_process := 2;
		2:
			
			IF gvl_axis.fbi_motionControler.out_flg_Done THEN
				gvl_axis.fbi_motionControler.in_flg_start := FALSE;
				var_process := 3;
			END_IF
		3:
			gvl_solv.fbi_ejector.in_var_vacMode := eP_ejeVacMode.break;
			gvl_solv.fbi_ejector.in_flg_run := TRUE;
			var_process := 4;
		4:
			IF gvl_solv.fbi_ejector.out_flg_Done THEN
				gvl_solv.fbi_ejector.in_flg_run := FALSE;
				var_process := 5;
			END_IF
		5:
			gvl_axis.fbi_motionControler.in_flg_start := FALSE;
			gvl_axis.fbi_motionControler.in_var_targetPosX := gvl_param.var_productInfo[gvl_param.var_currentProductID].teachPos.initial.x;
			gvl_axis.fbi_motionControler.in_var_targetPosY := gvl_param.var_productInfo[gvl_param.var_currentProductID].teachPos.remove.y;
			gvl_axis.fbi_motionControler.in_var_targetPosZ := gvl_param.var_productInfo[gvl_param.var_currentProductID].teachPos.initial.z;
			gvl_axis.fbi_motionControler.in_var_direction := eP_motionDirection.Z_X_Y;
			var_process := 6;
		6:
			gvl_axis.fbi_motionControler.in_flg_start := TRUE;
			var_process := 7;
		7:
			
			IF gvl_axis.fbi_motionControler.out_flg_Done THEN
				gvl_axis.fbi_motionControler.in_flg_start := FALSE;
				var_process := 8;
			END_IF
		8:
			gvl_auto.flg_pocketCountCheck := FALSE;
			trn_garbageDone := TRUE;
	END_CASE
END_IF
END_ACTION

ACTION moveToInitPos_active:
IF moveToInitPos._x AND moveToInitPos.x = FALSE THEN
	trn_moveToInitPosDone := FALSE;
	var_process := 0;
ELSIF moveToInitPos._x AND moveToInitPos.x THEN
	CASE var_process OF
		0:
			gvl_axis.fbi_motionControler.in_var_targetPosX := gvl_param.var_productInfo[gvl_param.var_currentProductID].teachPos.initial.x;
			gvl_axis.fbi_motionControler.in_var_targetPosY := gvl_param.var_productInfo[gvl_param.var_currentProductID].teachPos.initial.y;
			gvl_axis.fbi_motionControler.in_var_targetPosZ := gvl_param.var_productInfo[gvl_param.var_currentProductID].teachPos.initial.z;
			gvl_axis.fbi_motionControler.in_var_direction := eP_motionDirection.ZYX;
			var_process := 1;
		1:
			gvl_axis.fbi_motionControler.in_flg_start := TRUE;
			IF gvl_axis.fbi_motionControler.out_flg_Done THEN
				gvl_auto.flg_axisIsPcikingUp := FALSE;
				gvl_axis.fbi_motionControler.in_flg_start := FALSE;
				var_process := 2;
			END_IF
		2:
			gvl_auto.flg_sampling := FALSE;
			trn_moveToInitPosDone := TRUE;
	END_CASE
END_IF
END_ACTION

PROPERTY p_Init : bool
GET
p_init := THIS^.SFCInit;
END_GET
SET
THIS^.SFCInit := p_init;
END_SET
END_PROPERTY

ACTION pocketCheck_active:
IF pocketCheck._x AND pocketCheck.x = FALSE THEN
	trn_trayChange := FALSE;
	trn_notTrayChange := FALSE;
	flg_pocketIsNotFull := FALSE;
ELSIF pocketCheck._x AND pocketCheck.x THEN
	FOR var_i := 1 TO gvl_param.var_productInfo[gvl_param.var_currentProductID].cavQty BY 1 DO
		IF gvl_auto.pocketNo[var_i] < gvl_param.var_productInfo[gvl_param.var_currentProductID].pocketSumQty THEN
			flg_pocketIsNotFull := TRUE;
		END_IF
		IF var_i = gvl_param.var_productInfo[gvl_param.var_currentProductID].cavQty THEN
			trn_trayChange := NOT flg_pocketIsNotFull;
			trn_notTrayChange := flg_pocketIsNotFull;
		END_IF
	END_FOR
END_IF
END_ACTION

ACTION sample_active:
IF sample._x AND sample.x = FALSE THEN
	gvl_axis.fbi_motionControler.in_flg_start := FALSE;
	gvl_elecylinder.fbi_axisSample.in_flg_run := FALSE;
	gvl_error.flg_sample_windown_warning:= FALSE;
	gvl_solv.fbi_ejector.in_flg_run := FALSE;
	flg_axisXY_move_Sample_Done := FALSE;
	flg_axisSample_Done := FALSE;
	trn_sampleDone := FALSE;
	flg_allLensIsNotSet := FALSE;
	gvl_auto.flg_sampling := TRUE;
	fb_TON_delay.IN := FALSE;
	fb_TON_delay_error.IN:= FALSE;
	var_process := -1;
ELSIF sample._x AND sample.x THEN
	fb_TON_delay();
	fb_TON_delay_error(PT:=T#60S);
	CASE var_process OF
		-1:
			var_process:= 0;
		0:
			fb_TON_delay.PT:= T#5S;
			fb_TON_delay.IN:= TRUE;
			fb_TON_delay_error.IN:= TRUE;;
			flg_sampleCavCheck[gvl_auto.buf_cavNo] := TRUE;
			gvl_axis.fbi_motionControler.in_var_targetPosX := gvl_param.var_productInfo[gvl_param.var_currentProductID].teachPos.sample[gvl_auto.buf_cavNo].x;
			gvl_axis.fbi_motionControler.in_var_targetPosY := gvl_param.var_productInfo[gvl_param.var_currentProductID].teachPos.sample[gvl_auto.buf_cavNo].y;
			gvl_axis.fbi_motionControler.in_var_targetPosZ := gvl_param.var_productInfo[gvl_param.var_currentProductID].teachPos.initial.z;
			gvl_axis.fbi_motionControler.in_var_direction := eP_motionDirection.Y_X_Z;
			gvl_elecylinder.fbi_axisSample.in_var_moveMode := eP_eleMoveMode.eleB;
			IF fb_TON_delay.Q THEN
				gvl_error.flg_sample_windown_warning:= TRUE;
				gvl_visu.var_msg:="サンプル台が移動する為に扉を閉じてください。";
			END_IF
			IF fb_TON_delay_error.Q THEN
				gvl_error.flg_sample_windown_error:= TRUE;
				gvl_visu.var_msg:="扉が閉まらないでサンプル台が移動出来ないエラー";
			END_IF
			IF gvl_io.flg_frontSaftyDoor OR gvl_elecylinder.ref_axis_sample.input.in_flg_sensB THEN
				gvl_elecylinder.fbi_axisSample.in_flg_run := TRUE;
				gvl_axis.fbi_motionControler.in_flg_start := TRUE;
				gvl_error.flg_sample_windown_warning:= FALSE;
				fb_TON_delay_error.IN:= FALSE;
				fb_TON_delay.IN := FALSE;
				var_process := 1;
			END_IF
		1:
			IF gvl_elecylinder.fbi_axisSample.out_flg_Done THEN
				flg_axisSample_Done:= TRUE;
				gvl_elecylinder.fbi_axisSample.in_flg_run := FALSE;
			END_IF
			IF gvl_axis.fbi_motionControler.out_flg_Done THEN
				flg_axisXY_move_Sample_Done:= TRUE;
				gvl_axis.fbi_motionControler.in_flg_start := FALSE;
			END_IF
			IF flg_axisSample_Done AND flg_axisXY_move_Sample_Done THEN
				flg_axisSample_Done := FALSE;
				flg_axisXY_move_Sample_Done := FALSE;
				var_process := 2;
			END_IF
		2:
			gvl_axis.fbi_motionControler.in_flg_start := FALSE;
			gvl_axis.fbi_motionControler.in_var_targetPosX := gvl_param.var_productInfo[gvl_param.var_currentProductID].teachPos.sample[gvl_auto.buf_cavNo].X;
			gvl_axis.fbi_motionControler.in_var_targetPosY := gvl_param.var_productInfo[gvl_param.var_currentProductID].teachPos.sample[gvl_auto.buf_cavNo].y;
			gvl_axis.fbi_motionControler.in_var_targetPosZ := gvl_param.var_productInfo[gvl_param.var_currentProductID].teachPos.sample[gvl_auto.buf_cavNo].Z;
			gvl_axis.fbi_motionControler.in_var_direction := eP_motionDirection.Z_X_Y;
			fb_TON_delay.PT:= T#200MS;
			fb_TON_delay.IN:= TRUE;
			IF fb_TON_delay.Q THEN
				fb_TON_delay.IN:= FALSE;
				var_process := 3;
			END_IF
		3:
			gvl_axis.fbi_motionControler.in_flg_start := TRUE;
			var_process := 4;
		4:
			IF gvl_axis.fbi_motionControler.out_flg_Done THEN
				gvl_axis.fbi_motionControler.in_flg_start := FALSE;
				var_process := 5;
			END_IF
		5:
			gvl_solv.fbi_ejector.in_var_vacMode := eP_ejeVacMode.break;
			gvl_solv.fbi_ejector.in_flg_run := TRUE;
			var_process := 6;
		6:
			
			IF gvl_solv.fbi_ejector.out_flg_Done THEN
				gvl_solv.fbi_ejector.in_flg_run := FALSE;
				var_process := 7;
			END_IF	
		7:
			gvl_axis.fbi_motionControler.in_flg_start := FALSE;
			gvl_axis.fbi_motionControler.in_var_targetPosX := gvl_param.var_productInfo[gvl_param.var_currentProductID].teachPos.initial.x;
			gvl_axis.fbi_motionControler.in_var_targetPosY := gvl_param.var_productInfo[gvl_param.var_currentProductID].teachPos.sample[gvl_auto.buf_cavNo].y;
			gvl_axis.fbi_motionControler.in_var_targetPosZ := gvl_param.var_productInfo[gvl_param.var_currentProductID].teachPos.initial.z;
			gvl_axis.fbi_motionControler.in_var_direction := eP_motionDirection.Z_X_Y;
			var_process := 8;
		8:
			gvl_axis.fbi_motionControler.in_flg_start := TRUE;
			var_process := 9;
		9:
			
			IF gvl_axis.fbi_motionControler.out_flg_Done THEN
				gvl_axis.fbi_motionControler.in_flg_start := FALSE;
				var_process := 10;
			END_IF
		10:
			FOR var_i := 1 TO gvl_param.var_productInfo[gvl_param.var_currentProductID].cavQty BY 1 DO
				IF flg_sampleCavCheck[var_i] = FALSE THEN
					flg_allLensIsNotSet := TRUE;
				END_IF
				IF var_i = gvl_param.var_productInfo[gvl_param.var_currentProductID].cavQty THEN
					IF flg_allLensIsNotSet  = FALSE THEN
						flg_sampleIsBusy := FALSE;
						gvl_visu.flg_btn_sample := FALSE;
						var_process := 11;
					ELSE
						var_process := 20;
					END_IF
				END_IF
			END_FOR
		11:
			FOR var_i_clear := 1 TO gvl_param.var_productInfo[gvl_param.var_currentProductID].cavQty BY 1 DO
				flg_sampleCavCheck[var_i_clear] := FALSE;
				IF var_i_clear = gvl_param.var_productInfo[gvl_param.var_currentProductID].cavQty THEN
					var_process := 12;
				END_IF
			END_FOR
		12:
			fb_TON_delay.PT:= T#5S;
			fb_TON_delay.IN:= TRUE;
			fb_TON_delay_error.IN:= TRUE;
			flg_axisSample_Done := FALSE;
			flg_axisXY_move_Sample_Done := FALSE;
			gvl_elecylinder.fbi_axisSample.in_flg_run := FALSE;
			gvl_elecylinder.fbi_axisSample.in_var_moveMode := eP_eleMoveMode.eleA;
			gvl_axis.fbi_motionControler.in_flg_start := FALSE;
			gvl_axis.fbi_motionControler.in_var_targetPosX := gvl_param.var_productInfo[gvl_param.var_currentProductID].teachPos.initial.x;
			gvl_axis.fbi_motionControler.in_var_targetPosY := gvl_param.var_productInfo[gvl_param.var_currentProductID].teachPos.initial.y;
			gvl_axis.fbi_motionControler.in_var_targetPosZ := gvl_param.var_productInfo[gvl_param.var_currentProductID].teachPos.initial.z;
			gvl_axis.fbi_motionControler.in_var_direction := eP_motionDirection.Z_X_Y;
			IF fb_TON_delay.Q THEN
				gvl_error.flg_sample_windown_warning:= TRUE;
				gvl_visu.var_msg:="サンプル台が移動する為に扉を閉じてください。";
			END_IF
			IF fb_TON_delay_error.Q THEN
				gvl_error.flg_sample_windown_error:= TRUE;
				gvl_visu.var_msg:="扉が閉まらないでサンプル台が移動出来ないエラー";
			END_IF
			IF gvl_io.flg_frontSaftyDoor THEN
				gvl_elecylinder.fbi_axisSample.in_flg_run := TRUE;
				gvl_axis.fbi_motionControler.in_flg_start := TRUE;
				gvl_error.flg_sample_windown_warning:= FALSE;
				fb_TON_delay_error.IN:= FALSE;
				fb_TON_delay.IN := FALSE;
				var_process := 13;
			END_IF
		13:
			IF gvl_elecylinder.fbi_axisSample.out_flg_Done THEN
				flg_axisSample_Done:= TRUE;
				gvl_elecylinder.fbi_axisSample.in_flg_run := FALSE;
			END_IF
			IF gvl_axis.fbi_motionControler.out_flg_Done THEN
				flg_axisXY_move_Sample_Done:= TRUE;
				gvl_axis.fbi_motionControler.in_flg_start := FALSE;
			END_IF
			IF flg_axisSample_Done AND flg_axisXY_move_Sample_Done THEN
				flg_axisSample_Done := FALSE;
				flg_axisXY_move_Sample_Done := FALSE;
				var_process := 20;
			END_IF
		20:
			gvl_auto.flg_pocketCountCheck := FALSE;
			trn_sampleDone := TRUE;
	END_CASE
END_IF
END_ACTION

ACTION sampleTriger_active:
IF sampleTriger._x AND sampleTriger.x = FALSE THEN
	IF gvl_visu.flg_btn_sample AND gvl_param.var_productInfo[gvl_param.var_currentProductID].startCav = gvl_auto.buf_cavNo OR flg_sampleIsBusy THEN
		IF flg_sampleCavCheck[gvl_auto.buf_cavNo] THEN
			flg_sample_need := FALSE;
		END_IF
		flg_sampleIsBusy := TRUE;
	ELSE
		flg_sampleIsBusy := FALSE;
	END_IF
ELSIF sampleTriger._x AND sampleTriger.x THEN
	IF gvl_visu.flg_btn_sample AND gvl_param.var_productInfo[gvl_param.var_currentProductID].startCav = gvl_auto.buf_cavNo OR flg_sampleIsBusy THEN
		IF flg_sampleCavCheck[gvl_auto.buf_cavNo] THEN
			flg_sample_need := FALSE;
		END_IF
		flg_sampleIsBusy := TRUE;
	ELSE
		flg_sampleIsBusy := FALSE;
	END_IF
END_IF
END_ACTION

ACTION tray_active:
IF tray._x AND tray.x = FALSE THEN
	gvl_axis.fbi_motionControler.in_flg_start := FALSE;
	gvl_solv.fbi_ejector.in_flg_run := FALSE;
	trn_trayDone := FALSE;
	var_process := 0;
ELSIF tray._x AND tray.x THEN
	IF gvl_visu.var_dev_palletizingMode = FALSE THEN
			CASE var_process OF
				0:
					gvl_axis.fbi_motionControler.in_var_targetPosX := var_targetPosX;
					gvl_axis.fbi_motionControler.in_var_targetPosY := var_targetPosY;
					gvl_axis.fbi_motionControler.in_var_targetPosZ := var_targetPosZ;
					gvl_axis.fbi_motionControler.in_var_direction := eP_motionDirection.XYZ;
					var_process := 1;
				1:
					gvl_axis.fbi_motionControler.in_flg_start := TRUE;
					var_process := 2;
				2:

					IF gvl_axis.fbi_motionControler.out_flg_Done THEN
						gvl_axis.fbi_motionControler.in_flg_start := FALSE;
						var_process := 3;
					END_IF
					//vacuum error check
					IF gvl_axis.fbi_motionControler.out_flg_moveXYDone THEN
						gvl_error.flg_vacuum := NOT gvl_solv.ref_ejector.input.in_flg_sensVac;
					END_IF
				3:
					gvl_solv.fbi_ejector.in_var_vacMode := eP_ejeVacMode.break;
					gvl_auto.pocketNo[gvl_auto.buf_cavNo] := gvl_auto.pocketNo[gvl_auto.buf_cavNo] + 1;
					gvl_solv.fbi_ejector.in_flg_run := TRUE;
					var_process := 4;
				4:
					
					IF gvl_solv.fbi_ejector.out_flg_Done THEN
						gvl_solv.fbi_ejector.in_flg_run := FALSE;
						var_process := 5;
					END_IF
				5:
					gvl_auto.flg_pocketCountCheck := FALSE;
					trn_trayDone := TRUE;
			END_CASE
	ELSIF gvl_visu.var_dev_palletizingMode := TRUE THEN
			CASE var_process OF
				0:
					gvl_axis.fbi_motionControler.in_var_targetPosX := var_targetPosX + gvl_param.var_productInfo[gvl_param.var_currentProductID].teachPos.palletize.upperLower[gvl_param.var_currentTrayPos].cav[gvl_auto.buf_cavNo].teachingDetail.passingPos.x;
					gvl_axis.fbi_motionControler.in_var_targetPosY := var_targetPosY + gvl_param.var_productInfo[gvl_param.var_currentProductID].teachPos.palletize.upperLower[gvl_param.var_currentTrayPos].cav[gvl_auto.buf_cavNo].teachingDetail.passingPos.y;
					gvl_axis.fbi_motionControler.in_var_targetPosZ := var_targetPosZ + gvl_param.var_productInfo[gvl_param.var_currentProductID].teachPos.palletize.upperLower[gvl_param.var_currentTrayPos].cav[gvl_auto.buf_cavNo].teachingDetail.passingPos.z;
					gvl_axis.fbi_motionControler.in_var_direction := eP_motionDirection.XYZ;
					var_process := 1;
				1:
					gvl_axis.fbi_motionControler.in_flg_start := TRUE;
					var_process := 2;
				2:
					
					IF gvl_axis.fbi_motionControler.out_flg_Done THEN
						gvl_axis.fbi_motionControler.in_flg_start := FALSE;
						var_process := 3;
					END_IF
					//vacuum error check
					IF gvl_axis.fbi_motionControler.out_flg_moveXYDone THEN
						gvl_error.flg_vacuum := NOT gvl_solv.ref_ejector.input.in_flg_sensVac;
					END_IF
					
				3:
					gvl_axis.ref_x.Velocity := gvl_param.var_productInfo[gvl_param.var_currentProductID].teachPos.palletize.upperLower[gvl_param.var_currentTrayPos].cav[gvl_auto.buf_cavNo].teachingDetailVels.x.vel;
					gvl_axis.ref_y.Velocity := gvl_param.var_productInfo[gvl_param.var_currentProductID].teachPos.palletize.upperLower[gvl_param.var_currentTrayPos].cav[gvl_auto.buf_cavNo].teachingDetailVels.y.vel;
					gvl_axis.ref_z.Velocity := gvl_param.var_productInfo[gvl_param.var_currentProductID].teachPos.palletize.upperLower[gvl_param.var_currentTrayPos].cav[gvl_auto.buf_cavNo].teachingDetailVels.z.vel;
					gvl_axis.ref_x.Position := var_targetPosX + gvl_param.var_productInfo[gvl_param.var_currentProductID].teachPos.palletize.upperLower[gvl_param.var_currentTrayPos].cav[gvl_auto.buf_cavNo].teachingDetail.settingPOs.x;
					gvl_axis.ref_y.Position := var_targetPosY + gvl_param.var_productInfo[gvl_param.var_currentProductID].teachPos.palletize.upperLower[gvl_param.var_currentTrayPos].cav[gvl_auto.buf_cavNo].teachingDetail.settingPOs.y;
					gvl_axis.ref_z.Position := var_targetPosZ + gvl_param.var_productInfo[gvl_param.var_currentProductID].teachPos.palletize.upperLower[gvl_param.var_currentTrayPos].cav[gvl_auto.buf_cavNo].teachingDetail.settingPOs.z;
					var_process := 4;
				4:
					gvl_axis.ref_x.Execute := TRUE;
					gvl_axis.ref_y.Execute := TRUE;
					gvl_axis.ref_z.Execute := TRUE;
					var_process := 5;
			
				5:
					IF gvl_axis.fbi_mc_absX.Done AND gvl_axis.fbi_mc_absY.Done AND gvl_axis.fbi_mc_absZ.Done THEN
						var_process := 6;
					END_IF
				6:
					gvl_axis.ref_x.Execute := FALSE;
					gvl_axis.ref_y.Execute := FALSE;
					gvl_axis.ref_z.Execute := FALSE;
					gvl_solv.fbi_ejector.in_var_vacMode := eP_ejeVacMode.break;
					gvl_auto.pocketNo[gvl_auto.buf_cavNo] := gvl_auto.pocketNo[gvl_auto.buf_cavNo] + 1;
					gvl_solv.fbi_ejector.in_flg_run := TRUE;
					var_process := 7;
				7:
					
					IF gvl_solv.fbi_ejector.out_flg_Done THEN
						gvl_solv.fbi_ejector.in_flg_run := FALSE;
						var_process := 8;
					END_IF
				8:
					gvl_axis.ref_x.Velocity := gvl_param.var_productInfo[gvl_param.var_currentProductID].autoVels.x.vel;
					gvl_axis.ref_y.Velocity := gvl_param.var_productInfo[gvl_param.var_currentProductID].autoVels.y.vel;
					gvl_axis.ref_z.Velocity := gvl_param.var_productInfo[gvl_param.var_currentProductID].autoVels.z.vel;
					gvl_auto.flg_pocketCountCheck := FALSE;
					trn_trayDone := TRUE;
			END_CASE
	END_IF
END_IF
END_ACTION

ACTION trayChange_active:
IF trayChange._x AND trayChange.x = FALSE THEN
	trn_trayChangeDone := FALSE;
	fbi_exchangeTraySystem.in_flg_start := FALSE;
ELSIF trayChange._x AND trayChange.x THEN
	fbi_exchangeTraySystem.in_flg_start := gvl_visu.flg_btn_trayChangeDone;
	trn_trayChangeDone := NOT gvl_visu.flg_btn_trayChangeDone;
	IF gvl_auto.flg_trayChangeDone THEN
		FOR var_i := 0 TO 8 BY 1 DO
			gvl_auto.pocketNo[var_i] := 0;
			IF var_i = 8 THEN
				fbi_exchangeTraySystem.in_flg_start := FALSE;
				gvl_visu.flg_btn_trayChangeDone := FALSE;
				trn_trayChangeDone := TRUE;
			END_IF
		END_FOR
	END_IF
END_IF
fbi_exchangeTraySystem(
	var_ref_ele:= gvl_elecylinder.ref_axis_trayChange, 
	in_flg_run:= TRUE, 
	in_flg_start:= , 
	in_flg_pause:= NOT gvl_io.flg_frontSaftyDoor, 
	out_flg_run=> , 
	out_flg_busy=> , 
	out_flg_Done=> gvl_auto.flg_trayChangeDone, 
	out_flg_error=> );
END_ACTION

TRANSITION trn_closedCheck:
IF gvl_auto.autoModeStop AND gvl_auto.flg_transportClosed THEN
	trn_closedCheck := TRUE;
ELSE
	trn_closedCheck := FALSE;
END_IF
END_TRANSITION

ACTION waittingLens_active:
IF pickUpLens._x AND pickUpLens.x = FALSE THEN
	vacuumRetryTimer.IN := FALSE;
	gvl_auto.flg_VacuumRetry := FALSE;
	gvl_solv.fbi_ejector.in_var_vacMode := eP_ejeVacMode.halt;
	gvl_axis.fbi_motionControler.in_flg_start := FALSE;
	gvl_axis.fbi_motionControler.in_var_targetPosX := gvl_param.var_productInfo[gvl_param.var_currentProductID].teachPos.pickUp.x;
	gvl_axis.fbi_motionControler.in_var_targetPosY := gvl_param.var_productInfo[gvl_param.var_currentProductID].teachPos.pickUp.y;
	gvl_axis.fbi_motionControler.in_var_targetPosZ := gvl_param.var_productInfo[gvl_param.var_currentProductID].teachPos.pickUp.z;
	gvl_axis.fbi_motionControler.in_var_direction := eP_motionDirection.XYZ;
	trn_pickUpLensDone := FALSE;
	gvl_auto.flg_axisIsPcikingUp := FALSE;
	var_process := 0;
	fbi_vacuumRetry.in_flg_run := FALSE;
	gvl_auto.flg_sampling := FALSE;
ELSIF pickUpLens._x AND pickUpLens.x THEN

	CASE var_process OF
		0:
			IF gvl_auto.requirementToPickUpLens THEN
				IF gvl_visu.flg_btn_usingMeasurementSystem THEN
					IF NOT gvl_auto.flg_gm_eleIsDown THEN
						gvl_auto.flg_axisIsPcikingUp := TRUE;
						gvl_axis.fbi_motionControler.in_flg_start := TRUE;
						var_process := 1;
					END_IF
				ELSE
					gvl_axis.fbi_motionControler.in_flg_start := TRUE;
					var_process := 1;
				END_IF
			END_IF
		1:
			IF gvl_axis.fbi_motionControler.out_flg_Done THEN
				gvl_solv.fbi_ejector.in_flg_run := TRUE;
				gvl_axis.fbi_motionControler.in_flg_start := FALSE;
				var_process := 2;
			END_IF
		2:
			vacuumRetryTimer.IN := TRUE;
			IF vacuumRetryTimer.Q THEN
				var_process := 3;
			END_IF
		3:
			gvl_auto.lensVacuumDone := TRUE;
			IF gvl_auto.chuckopenDone THEN
				var_process := 4;
			END_IF
		4:
			gvl_axis.fbi_motionControler.in_flg_start := FALSE;
			gvl_axis.fbi_motionControler.in_var_targetPosX := gvl_param.var_productInfo[gvl_param.var_currentProductID].teachPos.initial.x;
			gvl_axis.fbi_motionControler.in_var_targetPosY := gvl_param.var_productInfo[gvl_param.var_currentProductID].teachPos.initial.y;
			gvl_axis.fbi_motionControler.in_var_targetPosZ := gvl_param.var_productInfo[gvl_param.var_currentProductID].teachPos.initial.z;
			gvl_axis.fbi_motionControler.in_var_direction := eP_motionDirection.ZYX;
			var_process := 5;
		5:
			gvl_axis.fbi_motionControler.in_flg_start := TRUE;
			var_process := 6;
		6:
			
			IF gvl_axis.fbi_motionControler.out_flg_Done THEN
				var_process := 7;
			END_IF
		7:
			IF NOT gvl_solv.ref_ejector.input.in_flg_sensVac THEN
				fbi_vacuumRetry.in_flg_run := TRUE;
				var_process := 8;
			ELSE
				var_process := 20;
			END_IF
		8:
			IF fbi_vacuumRetry.out_flg_Done THEN
				var_process := 20;
			ELSIF fbi_vacuumRetry.out_flg_faied THEN
				var_process := 10;
			END_IF
		10:
					
		20:	
			flg_sample_need:=TRUE;
			gvl_auto.pickUpLnesDone := TRUE;
			trn_pickUpLensDone := TRUE;
		
		END_CASE
END_IF
vacuumRetryTimer(IN:= , PT:=T#0.3S , Q=> , ET=> );
fbi_vacuumRetry(in_flg_run:= , out_flg_faied=> , out_flg_Done=> );
END_ACTION

END_FUNCTION_BLOCK

// ---- FBs/fb_exchangeTraySystem.TcPOU
FUNCTION_BLOCK fb_exchangeTraySystem
VAR_IN_OUT
	var_ref_ele : ref_ele_io;
END_VAR
VAR_INPUT
	in_flg_run : BOOL;
	in_flg_start : BOOL;
	in_flg_pause : BOOL;
END_VAR
VAR_OUTPUT
	out_flg_run : BOOL;
	out_flg_busy : BOOL;
	out_flg_Done : BOOL;
	out_flg_error : BOOL;
END_VAR
VAR
	fbi_ele_controler: fb_ele_controller;
	var_buf_moveMode : eP_eleMoveMode;
	flg_run: BOOL;
END_VAR
VAR // added by the converter: edge detectors and wires of the graphical bodies
    _rt1 : R_TRIG;
    _ft1, _ft2 : F_TRIG;
    _w1 : BOOL;
END_VAR

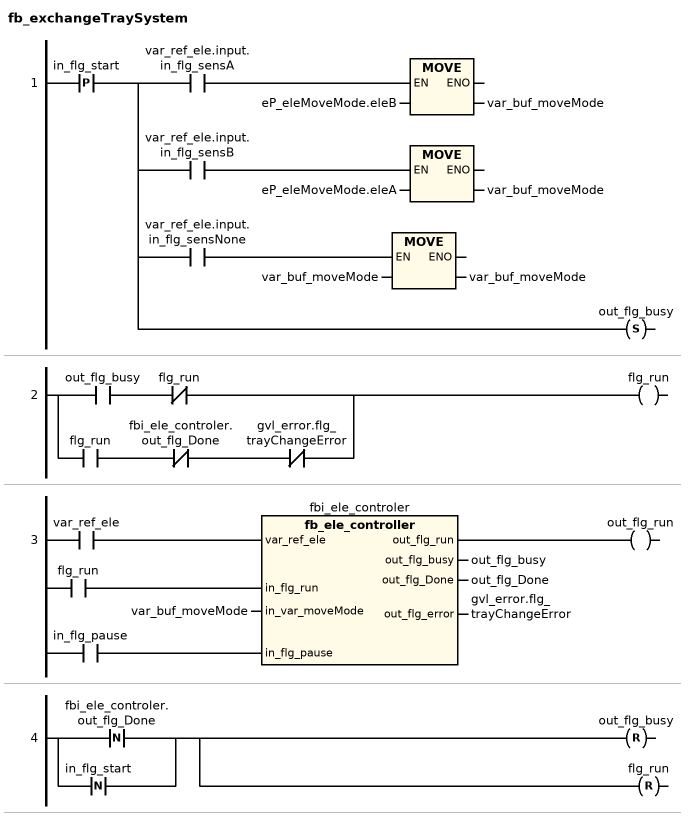
// NETWORK 1
_rt1(CLK := in_flg_start);
IF _rt1.Q AND var_ref_ele.input.in_flg_sensA THEN var_buf_moveMode := eP_eleMoveMode.eleB; END_IF
IF _rt1.Q AND var_ref_ele.input.in_flg_sensB THEN var_buf_moveMode := eP_eleMoveMode.eleA; END_IF
IF _rt1.Q AND var_ref_ele.input.in_flg_sensNone THEN var_buf_moveMode := var_buf_moveMode; END_IF
out_flg_busy S= _rt1.Q;

// NETWORK 2
flg_run := out_flg_busy AND NOT flg_run OR flg_run AND NOT fbi_ele_controler.out_flg_Done AND NOT gvl_error.flg_trayChangeError;

// NETWORK 3
fbi_ele_controler(
    var_ref_ele := var_ref_ele,
    in_flg_run := flg_run,
    in_var_moveMode := var_buf_moveMode,
    in_flg_pause := in_flg_pause,
    out_flg_busy => out_flg_busy,
    out_flg_Done => out_flg_Done,
    out_flg_error => gvl_error.flg_trayChangeError); // fb_ele_controller
out_flg_run := fbi_ele_controler.out_flg_run;

// NETWORK 4
_ft1(CLK := fbi_ele_controler.out_flg_Done);
_ft2(CLK := in_flg_start);
_w1 := _ft1.Q OR _ft2.Q;
out_flg_busy R= _w1;
flg_run R= _w1;

END_FUNCTION_BLOCK

// ---- FBs/fb_ele/fb_ele_controller.TcPOU
FUNCTION_BLOCK fb_ele_controller
VAR_IN_OUT
	var_ref_ele : ref_ele_io;
END_VAR
VAR_INPUT
	in_flg_run : BOOL;
	in_var_moveMode : eP_eleMovemode;
	in_flg_pause : BOOL;
END_VAR
VAR_OUTPUT
	out_flg_run : BOOL;
	out_flg_busy: BOOL;
	out_flg_Done: BOOL;
	out_flg_error : BOOL;
END_VAR
VAR
	var_buf_eleMoveMode: eP_eleMoveMode;
	flg_eleADone: BOOL;
	flg_eleBDone: BOOL;
	flg_eleStopDone: BOOL;
	fbi_timOut: TON;
	fb_TON_delay: TON;
END_VAR
VAR // added by the converter: edge detectors and wires of the graphical bodies
    _rt1, _rt2, _rt3, _rt4 : R_TRIG;
    _ft1, _ft2 : F_TRIG;
    _w1, _w2, _w3, _w4, _w5, _w6, _w7, _w8 : BOOL;
END_VAR

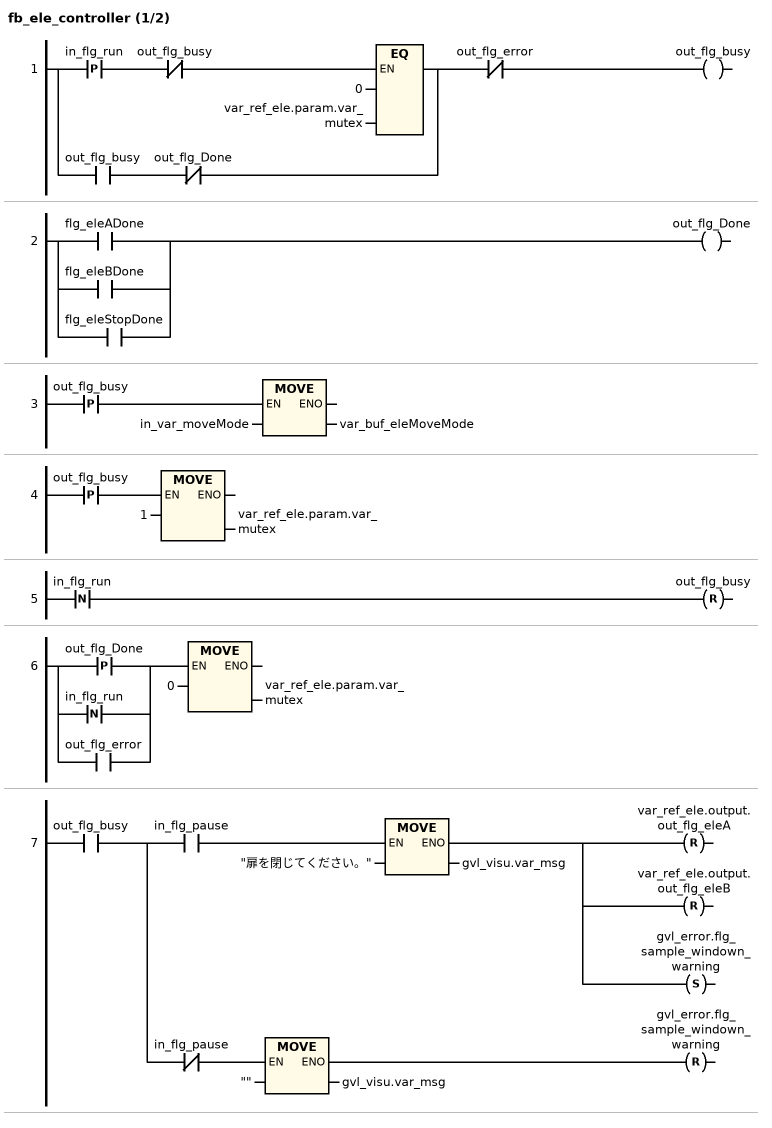
// NETWORK 1
_rt1(CLK := in_flg_run);
out_flg_busy := (_rt1.Q AND NOT out_flg_busy AND 0 = var_ref_ele.param.var_mutex OR out_flg_busy AND NOT out_flg_Done) AND NOT out_flg_error;

// NETWORK 2
out_flg_Done := flg_eleADone OR flg_eleBDone OR flg_eleStopDone;

// NETWORK 3
_rt2(CLK := out_flg_busy);
IF _rt2.Q THEN var_buf_eleMoveMode := in_var_moveMode; END_IF

// NETWORK 4
_rt3(CLK := out_flg_busy);
IF _rt3.Q THEN var_ref_ele.param.var_mutex := 1; END_IF

// NETWORK 5
_ft1(CLK := in_flg_run);
out_flg_busy R= _ft1.Q;

// NETWORK 6
_rt4(CLK := out_flg_Done);
_ft2(CLK := in_flg_run);
IF _rt4.Q OR _ft2.Q OR out_flg_error THEN var_ref_ele.param.var_mutex := 0; END_IF

// NETWORK 7
_w1 := out_flg_busy AND in_flg_pause;
IF _w1 THEN gvl_visu.var_msg := "扉を閉じてください。"; END_IF
var_ref_ele.output.out_flg_eleA R= _w1;
var_ref_ele.output.out_flg_eleB R= _w1;
gvl_error.flg_sample_windown_warning S= _w1;
_w2 := out_flg_busy AND NOT in_flg_pause;
IF _w2 THEN gvl_visu.var_msg := ""; END_IF
gvl_error.flg_sample_windown_warning R= _w2;

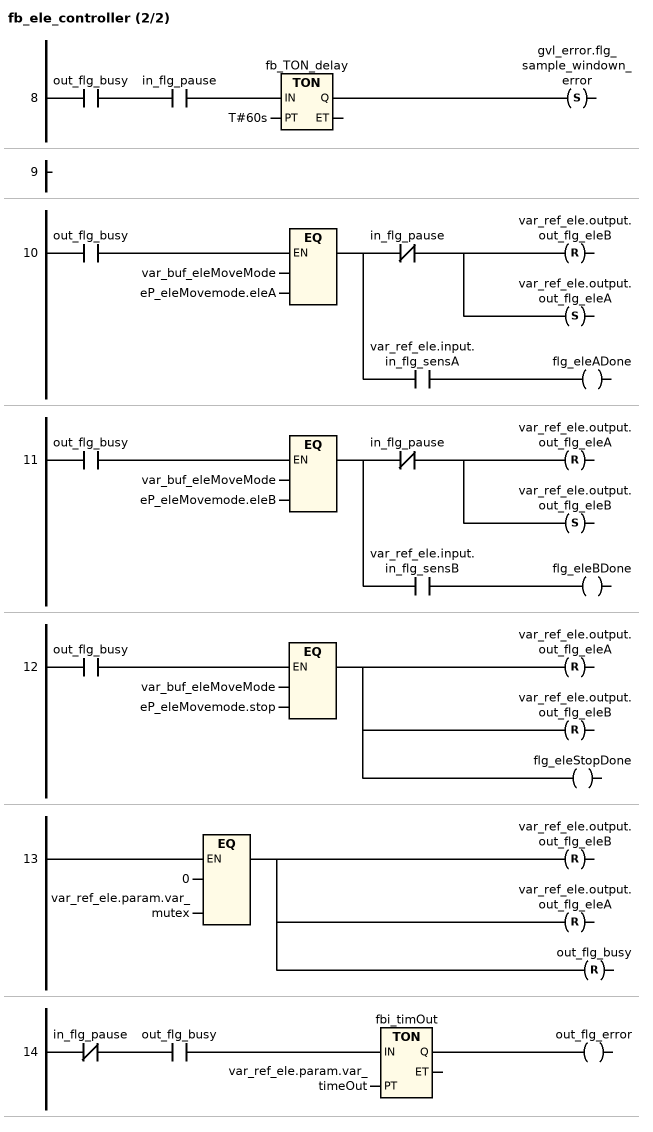
// NETWORK 8
fb_TON_delay(IN := out_flg_busy AND in_flg_pause, PT := T#60s); // TON
gvl_error.flg_sample_windown_error S= fb_TON_delay.Q;

// NETWORK 9

// NETWORK 10
_w3 := out_flg_busy AND var_buf_eleMoveMode = eP_eleMovemode.eleA;
_w4 := _w3 AND NOT in_flg_pause;
var_ref_ele.output.out_flg_eleB R= _w4;
var_ref_ele.output.out_flg_eleA S= _w4;
flg_eleADone := _w3 AND var_ref_ele.input.in_flg_sensA;

// NETWORK 11
_w5 := out_flg_busy AND var_buf_eleMoveMode = eP_eleMovemode.eleB;
_w6 := _w5 AND NOT in_flg_pause;
var_ref_ele.output.out_flg_eleA R= _w6;
var_ref_ele.output.out_flg_eleB S= _w6;
flg_eleBDone := _w5 AND var_ref_ele.input.in_flg_sensB;

// NETWORK 12
_w7 := out_flg_busy AND var_buf_eleMoveMode = eP_eleMovemode.stop;
var_ref_ele.output.out_flg_eleA R= _w7;
var_ref_ele.output.out_flg_eleB R= _w7;
flg_eleStopDone := _w7;

// NETWORK 13
_w8 := 0 = var_ref_ele.param.var_mutex;
var_ref_ele.output.out_flg_eleB R= _w8;
var_ref_ele.output.out_flg_eleA R= _w8;
out_flg_busy R= _w8;

// NETWORK 14
fbi_timOut(IN := NOT in_flg_pause AND out_flg_busy, PT := var_ref_ele.param.var_timeOut); // TON
out_flg_error := fbi_timOut.Q;

END_FUNCTION_BLOCK

// ---- FBs/fb_vacuumRetry.TcPOU
FUNCTION_BLOCK fb_vacuumRetry
VAR_INPUT
	in_flg_run: BOOL;
END_VAR
VAR_OUTPUT
	out_flg_faied: BOOL;
	out_flg_Done: BOOL;
END_VAR
VAR
	fbi_flg_run: R_TRIG;
	var_process: INT;
	var_retryTimes: INT;
	flg_chuckDone: BOOL;
	flg_pushDone: BOOL;
END_VAR

fbi_flg_run(CLK:= in_flg_run, Q=> );
IF fbi_flg_run.Q  THEN
	var_process := 1;
END_IF
IF NOT in_flg_run THEN
	out_flg_done := FALSE;
	out_flg_faied := FALSE;
	flg_chuckDone := FALSE;
	flg_pushDone := FALSE;
	var_retryTimes := 0;
END_IF
CASE var_process OF 
	1:
		gvl_axis.fbi_motionControler.in_flg_start := FALSE;
		gvl_axis.fbi_motionControler.in_var_targetPosX := gvl_param.var_productInfo[gvl_param.var_currentProductID].teachPos.pickUp.x;
		gvl_axis.fbi_motionControler.in_var_targetPosY := gvl_param.var_productInfo[gvl_param.var_currentProductID].teachPos.pickUp.y;
		gvl_axis.fbi_motionControler.in_var_targetPosZ := gvl_param.var_productInfo[gvl_param.var_currentProductID].teachPos.pickUp.z;
		gvl_axis.fbi_motionControler.in_var_direction := eP_motionDirection.XYZ;
		gvl_solv.fbi_chuck.in_flg_run := FALSE;
		gvl_solv.fbi_chuck.in_var_moveMode := eP_svMoveMode.svB;
		gvl_solv.fbi_push.in_flg_run := FALSE;
		gvl_solv.fbi_push.in_var_moveMode := eP_svMoveMode.svB;
		flg_chuckDone := FALSE;
		flg_pushDone := FALSE;
		var_process := 2;
	2:
		gvl_solv.fbi_push.in_flg_run := TRUE;
		gvl_solv.fbi_chuck.in_flg_run := TRUE;
		var_process := 3;
	3:
		IF gvl_solv.fbi_chuck.out_flg_Done THEN
			flg_chuckDone := TRUE;
		END_IF
		IF gvl_solv.fbi_push.out_flg_Done THEN
			flg_pushDone := TRUE;
		END_IF
		IF flg_pushDone AND flg_chuckDone THEN
			gvl_axis.fbi_motionControler.in_flg_start := TRUE;
			var_process := 4;
		END_IF
	4:
		IF gvl_axis.fbi_motionControler.out_flg_Done THEN
			gvl_axis.fbi_motionControler.in_flg_start := FALSE;
			var_process := 5;
		END_IF
	5:
		gvl_axis.fbi_motionControler.in_flg_start := FALSE;
		gvl_axis.fbi_motionControler.in_var_targetPosX := gvl_param.var_productInfo[gvl_param.var_currentProductID].teachPos.initial.x;
		gvl_axis.fbi_motionControler.in_var_targetPosY := gvl_param.var_productInfo[gvl_param.var_currentProductID].teachPos.initial.y;
		gvl_axis.fbi_motionControler.in_var_targetPosZ := gvl_param.var_productInfo[gvl_param.var_currentProductID].teachPos.initial.z;
		gvl_axis.fbi_motionControler.in_var_direction := eP_motionDirection.ZYX;
		gvl_solv.fbi_chuck.in_flg_run := FALSE;
		gvl_solv.fbi_chuck.in_var_moveMode := eP_svMoveMode.svA;
		gvl_solv.fbi_push.in_flg_run := FALSE;
		gvl_solv.fbi_push.in_var_moveMode := eP_svMoveMode.svA;
		flg_chuckDone := FALSE;
		flg_pushDone := FALSE;
		var_process := 6;
	6:
		gvl_solv.fbi_chuck.in_flg_run := TRUE;
		gvl_solv.fbi_push.in_flg_run := TRUE;
		IF gvl_solv.fbi_chuck.out_flg_Done THEN
			flg_chuckDone := TRUE;
		END_IF
		IF gvl_solv.fbi_push.out_flg_Done THEN
			flg_pushDone := TRUE;
		END_IF
		IF flg_pushDone AND flg_chuckDone THEN
			gvl_axis.fbi_motionControler.in_flg_start := TRUE;
			var_process := 7;
		END_IF
	7:
		IF gvl_axis.fbi_motionControler.out_flg_Done THEN
			gvl_axis.fbi_motionControler.in_flg_start := FALSE;
			var_process := 8;
		END_IF
	8:
		IF gvl_solv.ref_ejector.input.in_flg_sensVac THEN
			var_process := 20;
		ELSE
			var_process := 9;
		END_IF
	9:
		IF var_retryTimes < 3 THEN
			var_retryTimes := var_retryTimes + 1;
			var_process := 1;
		ELSE
			gvl_solv.fbi_ejector.in_flg_run := FALSE;
			gvl_solv.fbi_ejector.in_var_vacMode := eP_ejevacMode.vacON;
			var_process := 10;
		END_IF
	10:
		gvl_solv.fbi_ejector.in_flg_run := TRUE;
		var_process := 11;
	20:
	
		out_flg_Done := TRUE;
		var_process := 21;
	21:
		out_flg_Done := FALSE;
END_CASE

END_FUNCTION_BLOCK

// ---- FBs/gateMeasurementModule/fb_gm_measurementModule.TcPOU
FUNCTION_BLOCK fb_gm_measurementModule
VAR_INPUT
	SFCInit : BOOL;
END_VAR
VAR_OUTPUT
END_VAR
VAR
	trn_connectionCheckDone: BOOL;
	trn_wattingForLensDone: BOOL;
	flg_buf_gateLengthISSuccessed: BOOL;
	flg_buf_dummySignal: BOOL;
	trn_readCavDone: BOOL;
	fbi_getCav: fb_getCav;
	trn_chuckDone: BOOL;
	var_chuckCount: INT;
	trn_requestPickUpDone: BOOL;
	TON_data: TON;
	fbi_delayTimer: TON;
	trn_AddCountDone: BOOL;
	trn_lotStampDone: BOOL;
	var_process: INT;
	fbi_ton: TON;
	trn_LensCheckDone: BOOL;
	flg_SensorCheckDone: BOOL;
	flg_incjet_runned: BOOL;
END_VAR

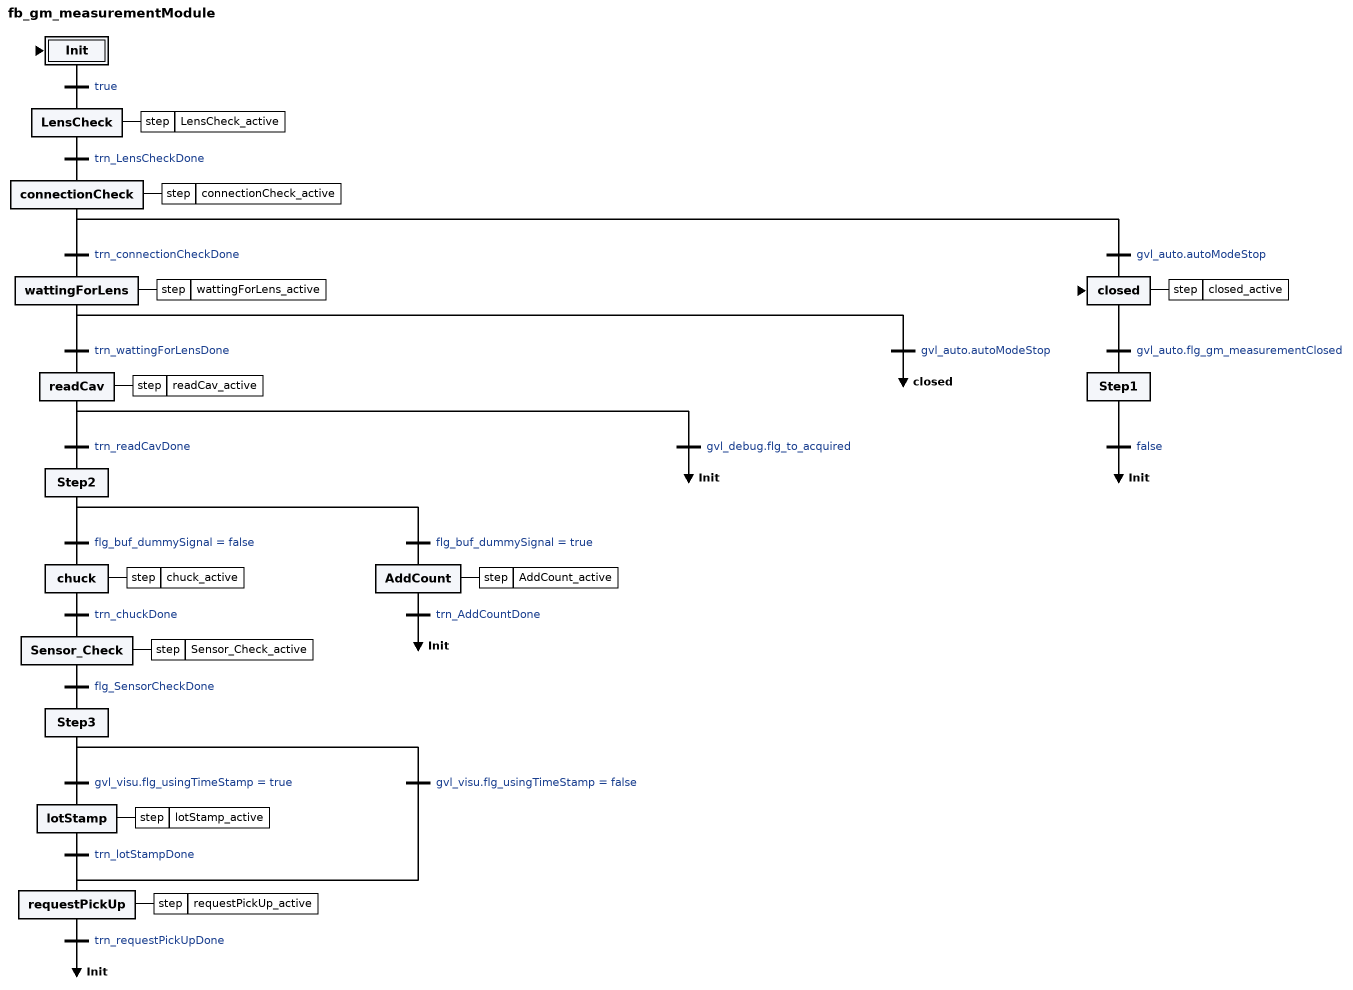
INITIAL_STEP Init:
END_STEP
TRANSITION FROM Init TO LensCheck
    := true;
END_TRANSITION
STEP LensCheck:
    LensCheck_active(N);  // step action
END_STEP
TRANSITION FROM LensCheck TO connectionCheck
    := trn_LensCheckDone;
END_TRANSITION
STEP connectionCheck:
    connectionCheck_active(N);  // step action
END_STEP
TRANSITION FROM connectionCheck TO wattingForLens
    := trn_connectionCheckDone;
END_TRANSITION
STEP wattingForLens:
    wattingForLens_active(N);  // step action
END_STEP
TRANSITION FROM wattingForLens TO readCav
    := trn_wattingForLensDone;
END_TRANSITION
TRANSITION FROM wattingForLens TO closed
    := gvl_auto.autoModeStop;
END_TRANSITION
TRANSITION FROM connectionCheck TO closed
    := gvl_auto.autoModeStop;
END_TRANSITION
STEP closed:
    closed_active(N);  // step action
END_STEP
TRANSITION FROM closed TO Step1
    := gvl_auto.flg_gm_measurementClosed;
END_TRANSITION
STEP Step1:
END_STEP
TRANSITION FROM Step1 TO Init
    := false;
END_TRANSITION
STEP readCav:
    readCav_active(N);  // step action
END_STEP
TRANSITION FROM readCav TO Step2
    := trn_readCavDone;
END_TRANSITION
TRANSITION FROM readCav TO Init
    := gvl_debug.flg_to_acquired;
END_TRANSITION
STEP Step2:
END_STEP
TRANSITION FROM Step2 TO chuck
    := flg_buf_dummySignal = false;
END_TRANSITION
TRANSITION FROM Step2 TO AddCount
    := flg_buf_dummySignal = true;
END_TRANSITION
STEP AddCount:
    AddCount_active(N);  // step action
END_STEP
TRANSITION FROM AddCount TO Init
    := trn_AddCountDone;
END_TRANSITION
STEP chuck:
    chuck_active(N);  // step action
END_STEP
TRANSITION FROM chuck TO Sensor_Check
    := trn_chuckDone;
END_TRANSITION
STEP Sensor_Check:
    Sensor_Check_active(N);  // step action
END_STEP
TRANSITION FROM Sensor_Check TO Step3
    := flg_SensorCheckDone;
END_TRANSITION
STEP Step3:
END_STEP
TRANSITION FROM Step3 TO lotStamp
    := gvl_visu.flg_usingTimeStamp = true;
END_TRANSITION
STEP lotStamp:
    lotStamp_active(N);  // step action
END_STEP
TRANSITION FROM lotStamp TO requestPickUp
    := trn_lotStampDone;
END_TRANSITION
TRANSITION FROM Step3 TO requestPickUp
    := gvl_visu.flg_usingTimeStamp = false;
END_TRANSITION
STEP requestPickUp:
    requestPickUp_active(N);  // step action
END_STEP
TRANSITION FROM requestPickUp TO Init
    := trn_requestPickUpDone;
END_TRANSITION

ACTION AddCount_active:
IF AddCount._x AND AddCount.x = FALSE THEN
	trn_AddCountDone := FALSE;
ELSIF AddCount._x AND AddCount.x THEN
	IF gvl_visu.flg_missingParts THEN
		gvl_gm.var_buf_measurementCav := gvl_auto.pocketNo[gvl_auto.buf_cavNo] + 1;
		trn_AddCountDone := TRUE;
	ELSE
		trn_AddCountDone := TRUE;
	END_IF
END_IF
END_ACTION

ACTION chuck_active:
IF chuck._x AND chuck.x = FALSE THEN
	TON_data.IN := FALSE;;
	trn_chuckDone := FALSE;
	gvl_solv.fbi_gm_chuck.in_flg_run := FALSE;
	gvl_solv.fbi_gm_push.in_flg_run := FALSE;
	gvl_auto.flg_gateData_Tx := FALSE;
	var_chuckCount := -11;
ELSIF chuck._x AND chuck.x THEN
	CASE var_chuckCount OF
		-11:
			IF gvl_param.var_productInfo[gvl_param.var_currentProductID].flg_mode_measurement THEN
				var_chuckCount := -10;
			ELSE
				var_chuckCount := 0;
			END_IF
		-10:
			gvl_solv.fbi_gm_push.in_var_moveMode := eP_svMoveMode.svB;
			gvl_solv.fbi_gm_push.in_flg_run := TRUE;
			var_chuckCount := -9;
		-9:
			IF gvl_solv.fbi_gm_push.out_flg_Done THEN
				gvl_solv.fbi_gm_push.in_flg_run := FALSE;
				var_chuckCount := -8;
			END_IF
		-8:
			gvl_solv.fbi_gm_push.in_var_moveMode := eP_svMoveMode.svA;
			gvl_solv.fbi_gm_push.in_flg_run := TRUE;
			var_chuckCount := -7;
		-7:
			IF gvl_solv.fbi_gm_push.out_flg_Done THEN
				gvl_solv.fbi_gm_push.in_flg_run := FALSE;
				var_chuckCount := -6;
			END_IF
		-6:
			gvl_solv.fbi_gm_chuck.in_var_moveMode := eP_svMoveMode.svB;
			gvl_solv.fbi_gm_chuck.in_flg_run := TRUE;
			var_chuckCount := -5;
		-5:
			IF gvl_solv.fbi_gm_chuck.out_flg_Done THEN
				gvl_solv.fbi_gm_chuck.in_flg_run := FALSE;
				var_chuckCount := -4;
			END_IF
		-4:
			gvl_solv.fbi_gm_push.in_var_moveMode := eP_svMoveMode.svB;
			gvl_solv.fbi_gm_push.in_flg_run := TRUE;
			var_chuckCount := -3;
		-3:
			IF gvl_solv.fbi_gm_push.out_flg_Done THEN
				gvl_solv.fbi_gm_push.in_flg_run := FALSE;
				var_chuckCount := 6;
			END_IF
		0:
			gvl_solv.fbi_gm_chuck.in_var_moveMode := eP_svMoveMode.svB;
			gvl_solv.fbi_gm_chuck.in_flg_run := TRUE;
			var_chuckCount := 1;
		1:
			
			IF gvl_solv.fbi_gm_chuck.out_flg_Done THEN
				gvl_solv.fbi_gm_chuck.in_flg_run := FALSE;
				var_chuckCount := 2;
			END_IF
		2:
			
			gvl_solv.fbi_gm_chuck.in_var_moveMode := eP_svMoveMode.svA;
			gvl_solv.fbi_gm_push.in_var_moveMode := eP_svMoveMode.svB;
			gvl_solv.fbi_gm_push.in_flg_run := TRUE;
			gvl_solv.fbi_gm_chuck.in_flg_run := TRUE;
			var_chuckCount := 3;
		3:
			IF gvl_solv.fbi_gm_push.out_flg_Done THEN
				gvl_solv.fbi_gm_push.in_flg_run := FALSE;
				gvl_solv.fbi_gm_chuck.in_flg_run := FALSE;
				var_chuckCount := 4;
			END_IF
		4:
			gvl_solv.fbi_gm_chuck.in_var_moveMode := eP_svMoveMode.svB;
			gvl_solv.fbi_gm_chuck.in_flg_run := TRUE;
			var_chuckCount := 5;
		5:
			IF gvl_solv.fbi_gm_chuck.out_flg_Done THEN
				gvl_solv.fbi_gm_chuck.in_flg_run := FALSE;
				var_chuckCount := 6;
			END_IF
		6:	
			TON_data.IN := TRUE;
			IF TON_data.Q THEN
				var_chuckCount := 7;
			END_IF
		7://gate measurement
			TON_data.IN := FALSE;
			IF gvl_io.flg_gm_fiberSens AND (gvl_io.var_gateLength > gvl_param.var_productInfo[gvl_param.var_currentProductID].gateLength_max OR gvl_io.var_gateLength < gvl_param.var_productInfo[gvl_param.var_currentProductID].gateLength_min) THEN
				gvl_gm.flg_gateLengthIsPassed := FALSE;
			ELSE
				gvl_gm.flg_gateLengthIsPassed := TRUE;
			END_IF
			gvl_auto.flg_gateData_Tx := TRUE;
			var_chuckCount := 8;
		8:
			gvl_solv.fbi_gm_chuck.in_flg_run := FALSE;
			var_chuckCount := 9;
		9:
			trn_chuckDone := TRUE;
	END_CASE
END_IF
TON_data(IN:= , PT:=T#200MS , Q=> , ET=> );
END_ACTION

ACTION closed_active:
IF closed._x AND closed.x = FALSE THEN
	gvl_auto.flg_gm_measurementClosed := FALSE;
ELSIF closed._x AND closed.x THEN
	gvl_io.flg_requestLens := FALSE;
	gvl_auto.flg_gm_measurementClosed := TRUE;
END_IF
END_ACTION

ACTION connectionCheck_active:
IF connectionCheck._x AND connectionCheck.x = FALSE THEN
	trn_connectionCheckDone:= FALSE;
	gvl_io.flg_requestLens := TRUE;
	var_process := 0;
ELSIF connectionCheck._x AND connectionCheck.x THEN
	CASE var_process OF
		0:
			IF gvl_io.flg_bitNumber0 
				AND gvl_io.flg_bitNumber1
				AND gvl_io.flg_bitNumber2
				AND gvl_io.flg_bitNumber3 OR gvl_debug.cavConecctSkip THEN
				trn_connectionCheckDone:= TRUE;
			END_IF
			IF NOT gvl_visu.flg_btn_vacSensOn THEN
				IF gvl_io.flg_gm_fiberSens THEN
					gvl_io.flg_requestLens := FALSE;
					IF((gvl_axis.axisX.NcToPlc.ActPos < gvl_visu.var_in_initialPos.x + 1) AND (gvl_axis.axisX.NcToPlc.ActPos > gvl_visu.var_in_initialPos.x - 1) AND NOT gvl_io.flg_fiberSens AND gvl_io.out_wire_ejectorVac ) THEN
						gvl_error.flg_gm_fiberSens := TRUE;
					END_IF
				END_IF
			END_IF
	END_CASE
	
END_IF
END_ACTION

ACTION LensCheck_active:
IF LensCheck._x AND LensCheck.x = FALSE THEN
	trn_LensCheckDone := FALSE;
	gvl_debug.flg_to_demand:= FALSE;
ELSIF LensCheck._x AND LensCheck.x THEN
	IF gvl_debug.out_busy THEN
		trn_LensCheckDone := TRUE;
	ELSE
		IF gvl_io.flg_gm_fiberSens THEN
			gvl_error.flg_gm_fiberSens := TRUE;	
		ELSE
			trn_LensCheckDone := TRUE;
		END_IF	
	END_IF
END_IF
END_ACTION

ACTION lotStamp_active:
IF lotStamp._x AND lotStamp.x = FALSE THEN
	trn_lotStampDone := FALSE;
	var_process := 0;
	fbi_ton.IN := FALSE;
	flg_incjet_runned:= FALSE;
ELSIF lotStamp._x AND lotStamp.x THEN
	CASE var_process OF
		0:
			fbi_ton.PT:= T#5S;
			fbi_ton.IN := TRUE;
			gvl_error.flg_incjet := fbi_ton.Q;
			gvl_gm.var_incjetInfo.flg_denyStamp := gvl_io.flg_gm_fiberSens;
			IF gvl_gm.var_incjetInfo.flg_stampReady THEN
				var_process := 1;
			END_IF
		1:
			fbi_ton.IN := FALSE;
			gvl_solv.fbi_gm_stamp.in_flg_run := FALSE;
			gvl_solv.fbi_gm_stamp.in_var_moveMode := eP_svMoveMode.svB;
			var_process := 2;
			
		2:
			gvl_solv.fbi_gm_stamp.in_flg_run := TRUE;
			var_process := 3;
		3:
			IF gvl_gm.var_incjetInfo.flg_stampRun THEN
				flg_incjet_runned:= TRUE;
			END_IF
			IF gvl_solv.fbi_gm_stamp.out_flg_Done THEN
				gvl_solv.fbi_gm_stamp.in_flg_run := FALSE;
				var_process := 4;
			END_IF
		4:
			fbi_ton.PT:= T#0.2S;
			fbi_ton.IN := TRUE;
			IF gvl_gm.var_incjetInfo.flg_stampRun THEN
				flg_incjet_runned:= TRUE;
			END_IF
			IF fbi_ton.Q THEN
				var_process := 5;
			END_IF
		5:
			IF flg_incjet_runned OR NOT gvl_gm.var_incjetInfo.flg_denyStamp THEN
				var_process := 6;
			ELSE
				gvl_error.flg_incjet:= TRUE;
			END_IF
		6:
			fbi_ton.IN := FALSE;
			gvl_solv.fbi_gm_stamp.in_var_moveMode := eP_svMoveMode.svA;
			gvl_solv.fbi_gm_stamp.in_flg_run := TRUE;
			var_process := 7;
		7:
			IF gvl_solv.fbi_gm_stamp.out_flg_Done THEN
				gvl_solv.fbi_gm_stamp.in_flg_run := FALSE;
				var_process := 8;
			END_IF
		8:
			flg_incjet_runned:= FALSE;
			gvl_gm.var_incjetInfo.flg_denyStamp := FALSE;
			trn_lotStampDone := TRUE;
	END_CASE
END_IF
fbi_ton(IN:= , PT:= , Q=> , ET=> );
END_ACTION

ACTION readCav_active:
IF readCav._x AND readCav.x = FALSE THEN
	trn_readCavDone := FALSE;
	THIS^.fbi_getCav();
	fbi_getCav.in_flg_run := FALSE;
	fbi_delayTimer.IN := FALSE;
ELSIF readCav._x AND readCav.x THEN
	THIS^.fbi_getCav();
	fbi_delayTimer.IN := TRUE;
	THIS^.fbi_getCav.in_flg_run := fbi_delayTimer.Q;
	IF gvl_debug.flg_debug_run THEN
		gvl_gm.var_buf_measurementCav := gvl_debug.var_cav;
		IF NOT (gvl_debug.flg_check_quality AND gvl_debug.flg_to_measurement) THEN
			trn_readCavDone := TRUE;
		END_IF
	ELSE
		IF THIS^.fbi_getCav.out_flg_Done THEN
			gvl_gm.var_buf_measurementCav := THIS^.fbi_getCav.out_var_cav;
			IF gvl_debug.flg_check_quality AND gvl_debug.flg_to_measurement THEN
				gvl_debug.flg_to_demand:= TRUE;
			ELSE
				trn_readCavDone := TRUE;
			END_IF
		ELSIF THIS^.fbi_getCav.out_flg_error THEN
			gvl_auto.cavNo := 0;
			IF gvl_debug.flg_check_quality AND gvl_debug.flg_to_measurement THEN
				gvl_debug.flg_to_demand:= TRUE;
			ELSE
				trn_readCavDone := TRUE;
			END_IF
		END_IF
	END_IF	
	
END_IF
fbi_delayTimer(IN:= , PT:=T#100MS , Q=> , ET=> );
END_ACTION

ACTION requestPickUp_active:
IF requestPickUp._x AND requestPickUp.x = FALSE THEN
	gvl_gm.flg_lensPickUpDone := FALSE;
	gvl_gm.flg_requestPickup := FALSE;
	trn_requestPickUpDone := false;
ELSIF requestPickUp._x AND requestPickUp.x THEN
	IF gvl_gm.flg_lensPickUpDone THEN
		gvl_gm.flg_requestPickup := FALSE;
		trn_requestPickUpDone := TRUE;
	ELSE
		gvl_gm.flg_requestPickup := TRUE;
	END_IF
END_IF
END_ACTION

ACTION Sensor_Check_active:
IF Sensor_Check._x AND Sensor_Check.x = FALSE THEN
	flg_SensorCheckDone := FALSE;
ELSIF Sensor_Check._x AND Sensor_Check.x THEN
	IF gvl_visu.flg_btn_vacSensOn THEN
		flg_SensorCheckDone:= TRUE;
	ELSE
		IF gvl_io.flg_gm_fiberSens THEN
			flg_SensorCheckDone:= TRUE;
		ELSE
			IF((gvl_axis.axisX.NcToPlc.ActPos < gvl_visu.var_in_initialPos.x + 1) AND (gvl_axis.axisX.NcToPlc.ActPos > gvl_visu.var_in_initialPos.x - 1) AND NOT gvl_io.flg_fiberSens AND gvl_io.out_wire_ejectorVac ) THEN
				gvl_error.flg_gm_fiberSens := TRUE;
			END_IF
		END_IF
	END_IF
END_IF
END_ACTION

ACTION wattingForLens_active:
IF wattingForLens._x AND wattingForLens.x = FALSE THEN
	trn_wattingForLensDone := FALSE;
	flg_buf_gateLengthISSuccessed := FALSE;
	flg_buf_dummySignal := FALSE;
ELSIF wattingForLens._x AND wattingForLens.x THEN
	//gate
	IF gvl_IO.flg_gateLengthIsSuccessed  THEN
		flg_buf_gateLengthISSuccessed := TRUE;
	END_IF
	//dummy signal
	IF gvl_io.flg_dummySiganl THEN
		flg_buf_dummySignal := TRUE;
	END_IF
	//lens set done
	IF gvl_debug.out_busy THEN
		IF gvl_visu.flg_btn_lensSetDone OR gvl_visu.flg_btn_vacSensOn THEN
			gvl_io.flg_requestLens := FALSE;
			trn_wattingForLensDone := TRUE;
		END_IF
	ELSE
		IF gvl_io.flg_lensSetDone THEN
			gvl_io.flg_requestLens := FALSE; 
			trn_wattingForLensDone := TRUE;
		END_IF
	END_IF
END_IF
END_ACTION

END_FUNCTION_BLOCK

// ---- FBs/gateMeasurementModule/fb_gm_transport.TcPOU
FUNCTION_BLOCK fb_gm_transport
VAR_INPUT
END_VAR
VAR_OUTPUT
END_VAR
VAR
	SFCInit : bool;
	trn_lensPickUpDone: BOOL;
	trn_transportDone: BOOL;
	trn_lensSetDone: BOOL;
	var_process: INT;
	trn_homeDone: BOOL;
	trn_closeCheckDone: BOOL;
	trn_waittingLensDone: BOOL;
	retryTimer: TON;
	var_retryTimes: INT;
END_VAR

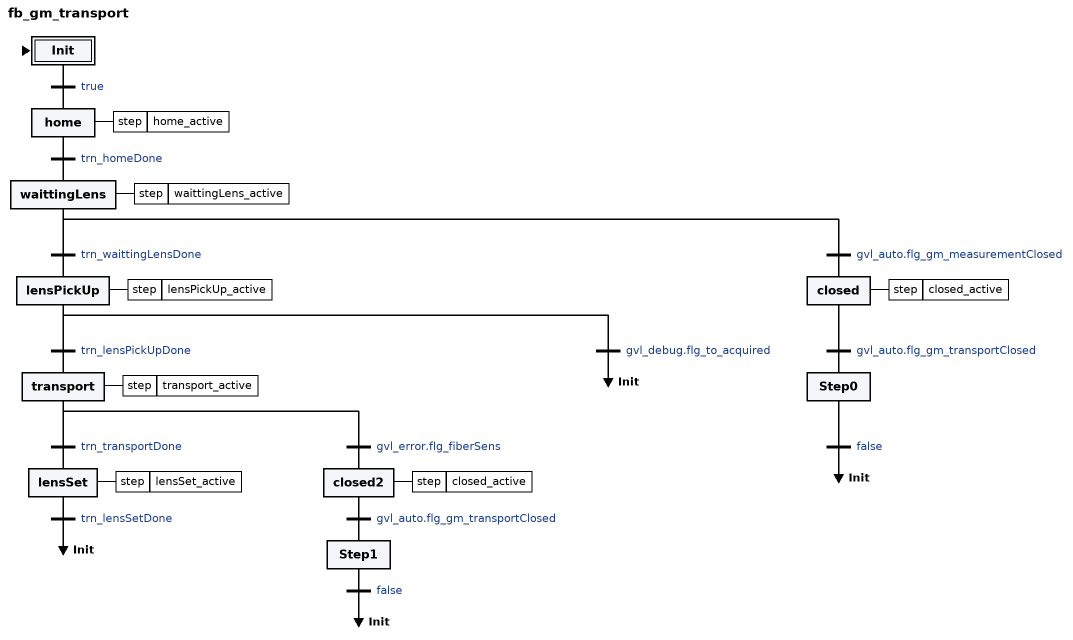
INITIAL_STEP Init:
END_STEP
TRANSITION FROM Init TO home
    := true;
END_TRANSITION
STEP home:
    home_active(N);  // step action
END_STEP
TRANSITION FROM home TO waittingLens
    := trn_homeDone;
END_TRANSITION
STEP waittingLens:
    waittingLens_active(N);  // step action
END_STEP
TRANSITION FROM waittingLens TO lensPickUp
    := trn_waittingLensDone;
END_TRANSITION
STEP lensPickUp:
    lensPickUp_active(N);  // step action
END_STEP
TRANSITION FROM lensPickUp TO transport
    := trn_lensPickUpDone;
END_TRANSITION
TRANSITION FROM lensPickUp TO Init
    := gvl_debug.flg_to_acquired;
END_TRANSITION
TRANSITION FROM waittingLens TO closed
    := gvl_auto.flg_gm_measurementClosed;
END_TRANSITION
STEP closed:
    closed_active(N);  // step action
END_STEP
TRANSITION FROM closed TO Step0
    := gvl_auto.flg_gm_transportClosed;
END_TRANSITION
STEP Step0:
END_STEP
TRANSITION FROM Step0 TO Init
    := false;
END_TRANSITION
STEP transport:
    transport_active(N);  // step action
END_STEP
TRANSITION FROM transport TO lensSet
    := trn_transportDone;
END_TRANSITION
STEP lensSet:
    lensSet_active(N);  // step action
END_STEP
TRANSITION FROM lensSet TO Init
    := trn_lensSetDone;
END_TRANSITION
TRANSITION FROM transport TO closed2
    := gvl_error.flg_fiberSens;
END_TRANSITION
STEP closed2:
    closed_active(N);  // step action
END_STEP
TRANSITION FROM closed2 TO Step1
    := gvl_auto.flg_gm_transportClosed;
END_TRANSITION
STEP Step1:
END_STEP
TRANSITION FROM Step1 TO Init
    := false;
END_TRANSITION

ACTION closed_active:
IF closed._x AND closed.x = FALSE THEN
	gvl_auto.flg_gm_transportClosed := FALSE;
ELSIF closed._x AND closed.x THEN
	gvl_auto.flg_gm_transportClosed := TRUE;
END_IF
END_ACTION

ACTION home_active:
IF home._x AND home.x = FALSE THEN
	var_process := 0;
	trn_homeDone := FALSE;
	gvl_debug.flg_to_demand:= FALSE;
ELSIF home._x AND home.x THEN
	CASE var_process OF 
		0:
			gvl_elecylinder.fbi_gm_axisPickUp.in_flg_run := FALSE;
			gvl_elecylinder.fbi_gm_axisPickUp.in_var_moveMode := eP_eleMoveMode.eleA;
			gvl_elecylinder.fbi_gm_axisTransport.in_flg_run := FALSE;
			gvl_elecylinder.fbi_gm_axisTransport.in_var_moveMode := eP_eleMoveMode.eleA;
			gvl_axis.ref_r.Execute := FALSE;
			gvl_axis.ref_r.Position := gvl_param.var_productInfo[gvl_param.var_currentProductID].teachPos.gm_rotary.origin;
			var_process := 1;
		1:
			gvl_elecylinder.fbi_gm_axisPickUp.in_flg_run := TRUE;
			gvl_elecylinder.fbi_gm_axisTransport.in_flg_run := TRUE;
			var_process := 2;
		2:
			IF gvl_elecylinder.ref_gm_axisPickUp.input.in_flg_sensA AND gvl_elecylinder.ref_gm_axisTransport.input.in_flg_sensA THEN
				gvl_elecylinder.fbi_gm_axisPickUp.in_flg_run := FALSE;
				gvl_elecylinder.fbi_gm_axisTransport.in_flg_run := FALSE;
				var_process := 3;
			END_IF
		3:
			gvl_solv.fbi_gm_pickup.in_flg_run := FALSE;
			gvl_solv.fbi_gm_pickup.in_var_moveMode := eP_svMoveMode.svA;
			var_process := 4;
		4:
			gvl_solv.fbi_gm_pickup.in_flg_run := TRUE;
			IF gvl_solv.ref_gm_pickUp.in.in_flg_sensA  THEN
				var_process := 5;
			END_IF
		5:
			gvl_auto.flg_gm_eleIsDown := FALSE;
			gvl_axis.ref_r.Execute := TRUE;
			IF gvl_axis.ref_r.Done THEN
				gvl_axis.ref_r.Execute := FALSE;
				var_process :=6;
			END_IF
		6:
			gvl_solv.fbi_gm_rotary.in_flg_run := FALSE;
			gvl_solv.fbi_gm_rotary.in_var_moveMode := eP_svMoveMode.svA;
			var_process := 7;
		7:
			gvl_solv.fbi_gm_rotary.in_flg_run := TRUE;
			IF gvl_solv.ref_gm_rotary.in.in_flg_sensA THEN
				var_process := 8;
			END_IF
		8:	
				trn_homeDone := TRUE;			
	END_CASE
END_IF
END_ACTION

ACTION lensPickUp_active:
IF lensPickUp._x AND lensPickUp.x = FALSE THEN
	gvl_axis.ref_r.Execute := FALSE;
	retryTimer.IN := FALSE;
	var_process := 0;
	var_retryTimes := 0;
	trn_lensPickUpDone := FALSE;
	gvl_auto.flg_gm_VacuumRetry := FALSE;
	gvl_solv.fbi_gm_ejector.in_flg_run := FALSE;
	gvl_solv.fbi_gm_pickup.in_flg_run := FALSE;
	gvl_solv.fbi_gm_rotary.in_flg_run := FALSE;
	gvl_elecylinder.fbi_gm_axisPickUp.in_flg_run := FALSE;
	gvl_axis.ref_r.Execute := FALSE;
ELSIF lensPickUp._x AND lensPickUp.x THEN
	CASE var_process OF 
		0:
			gvl_axis.ref_r.Position := gvl_param.var_productInfo[gvl_param.var_currentProductID].teachPos.gm_rotary.pickUp;
			gvl_axis.ref_r.Execute := TRUE;
			gvl_solv.fbi_gm_ejector.in_var_vacMode := eP_ejeVacMode.vacON;
			gvl_solv.fbi_gm_ejector.in_flg_run := TRUE;
			var_process := 1;
		1://axis theta move to pick up position
			gvl_solv.fbi_gm_ejector.in_flg_run := FALSE;
			IF gvl_axis.ref_r.Done THEN
				gvl_axis.ref_r.Execute := FALSE;
				var_process := 2;
			END_IF
		2:
			IF gvl_solv.ref_gm_ejctor.input.in_flg_sensVac THEN
				var_process := 3;
			END_IF
		3:
			gvl_solv.fbi_gm_chuck.in_var_moveMode := eP_svMoveMode.svA;
			gvl_solv.fbi_gm_push.in_var_moveMode := eP_svMoveMode.svA;
			gvl_solv.fbi_gm_chuck.in_flg_run := TRUE;
			gvl_solv.fbi_gm_push.in_flg_run := TRUE;
			var_process := 4;
		4:
			IF gvl_solv.ref_gm_chuck.in.in_flg_sensA AND gvl_solv.ref_gm_push.in.in_flg_sensA THEN
				gvl_solv.fbi_gm_chuck.in_flg_run := FALSE;
				gvl_solv.fbi_gm_push.in_flg_run := FALSE;
				var_process := 5;
			END_IF
		5:
			gvl_solv.fbi_gm_pickup.in_var_moveMode := eP_svMoveMode.svB;
			gvl_solv.fbi_gm_pickup.in_flg_run := TRUE;
			var_process := 6;
		6:
			IF gvl_solv.fbi_gm_pickup.out_flg_Done THEN
				gvl_solv.fbi_gm_pickup.in_flg_run := FALSE;
				var_process := 7;
			END_IF
		7:
			gvl_axis.ref_r.Position := gvl_param.var_productInfo[gvl_param.var_currentProductID].teachPos.gm_rotary.set;
			gvl_axis.ref_r.Execute := TRUE;
			var_process := 8;
		8:
			IF gvl_axis.ref_r.Done THEN
				gvl_axis.ref_r.Execute := FALSE;
				var_process := 9;	
			END_IF
		9:
			gvl_solv.fbi_gm_pickup.in_var_moveMode := eP_svMoveMode.svA;
			gvl_solv.fbi_gm_pickup.in_flg_run := TRUE;
			var_process := 10;
		10:
			IF gvl_solv.fbi_gm_pickup.out_flg_Done THEN
				gvl_solv.fbi_gm_pickup.in_flg_run := FALSE;
				var_process := 11;
			END_IF
		11:
			gvl_solv.fbi_gm_rotary.in_flg_run := FALSE;
			gvl_solv.fbi_gm_rotary.in_var_moveMode := eP_svMoveMode.svB;
			var_process:= 12;
		12:
			gvl_solv.fbi_gm_rotary.in_flg_run := TRUE;
			var_process := 13;
		13:
			IF gvl_solv.fbi_gm_rotary.out_flg_Done THEN
				gvl_solv.fbi_gm_rotary.in_flg_run := FALSE;
				var_process := 14;
			END_IF
		14:
			gvl_solv.fbi_gm_pickup.in_var_moveMode := eP_svMoveMode.svB;
			gvl_solv.fbi_gm_pickup.in_flg_run := TRUE;
			var_process := 15;
		15:
			IF gvl_solv.fbi_gm_pickup.out_flg_Done THEN
				gvl_solv.fbi_gm_pickup.in_flg_run := FALSE;
				var_process := 16;
			END_IF
		16:
			gvl_gm.flg_lensPickUpDone := TRUE;
			gvl_gm.var_buf_tranportCav := gvl_gm.var_buf_measurementCav;
			gvl_gm.flg_buf_gateLengthIsPassed := gvl_gm.flg_gateLengthIsPassed;
			var_process := 17;
		17:
			IF gvl_gm.flg_lensRequest AND NOT gvl_auto.flg_axisIsPcikingUp THEN
				IF gvl_debug.flg_check_quality AND gvl_debug.flg_to_stocker THEN
					gvl_debug.flg_to_demand:= TRUE;
				ELSE
					trn_lensPickUpDone := TRUE;		
				END_IF
			END_IF		
	END_CASE
END_IF
END_ACTION

ACTION lensSet_active:
IF lensSet._x AND lensSet.x = FALSE THEN
	trn_lensSetDone := FALSE;
	var_process := 0;
ELSIF lensSet._x AND lensSet.x THEN
	CASE var_process OF
		0:
			gvl_solv.fbi_gm_ejector.in_var_vacMode := eP_ejeVacMode.break;
			gvl_solv.fbi_gm_ejector.in_flg_run := FALSE;
			gvl_elecylinder.fbi_gm_axisPickUp.in_var_moveMode := eP_eleMoveMode.eleA;
			gvl_elecylinder.fbi_gm_axisPickUp.in_flg_run := FALSE;
			var_process := 1;
		1:
			gvl_solv.fbi_gm_ejector.in_flg_run := TRUE;
			IF gvl_solv.fbi_gm_ejector.out_flg_Done THEN
				gvl_solv.fbi_gm_ejector.in_flg_run := FALSE;
				var_process := 2;
			END_IF
		2:
			gvl_elecylinder.fbi_gm_axisPickUp.in_flg_run := TRUE;
			IF gvl_elecylinder.fbi_gm_axisPickUp.out_flg_Done THEN
				gvl_elecylinder.fbi_gm_axisPickUp.in_flg_run := FALSE;
				var_process := 3;
			END_IF
		3:
			gvl_gm.flg_lensSetDoneFromGM := TRUE;
			trn_lensSetDone := TRUE;
	END_CASE
END_IF
END_ACTION

PROPERTY p_Init : bool
GET
p_init := THIS^.SFCInit;
END_GET
SET
THIS^.SFCInit := p_init;
END_SET
END_PROPERTY

ACTION transport_active:
IF transport._x AND transport.x = FALSE THEN
	var_process := 0;
	trn_transportDone := FALSE;
	gvl_elecylinder.fbi_gm_axisTransport.in_flg_run := FALSE;
	gvl_elecylinder.fbi_gm_axisTransport.in_var_moveMode := eP_eleMoveMode.eleB;
	gvl_elecylinder.fbi_gm_axisPickUp.in_flg_run := FALSE;
	gvl_elecylinder.fbi_gm_axisPickUp.in_var_moveMode := eP_eleMoveMode.eleB;
	gvl_solv.fbi_gm_pickup.in_flg_run := FALSE;
	gvl_solv.fbi_gm_pickup.in_var_moveMode := eP_svMoveMode.svB;
	gvl_solv.fbi_gm_rotary.in_flg_run := FALSE;
	//gvl_solv.fbi_gm_rotary.in_var_moveMode := eP_svMoveMode.svB;
ELSIF transport._x AND transport.x THEN
	CASE var_process OF
		0:
			IF NOT gvl_auto.flg_axisIsPcikingUp THEN
				//var_process := 1;
				var_process := 3;
			END_IF
		//1:
			//gvl_solv.fbi_gm_rotary.in_flg_run := TRUE;
			//var_process := 2;
		//2:
			//IF gvl_solv.fbi_gm_rotary.out_flg_Done THEN
				//gvl_solv.fbi_gm_rotary.in_flg_run := FALSE;
				//var_process := 3;
			//END_IF
		3:
			IF NOT gvl_io.flg_fiberSens THEN
				gvl_auto.flg_gm_eleIsDown := TRUE;
				gvl_elecylinder.fbi_gm_axisTransport.in_flg_run := TRUE;
				gvl_elecylinder.fbi_gm_axisPickUp.in_flg_run := TRUE;
				gvl_solv.fbi_gm_pickup.in_flg_run := TRUE;
				var_process := 4;
			ELSE
				gvl_error.flg_fiberSens:= TRUE;
			END_IF
		4:
			IF gvl_elecylinder.fbi_gm_axisTransport.out_flg_Done THEN
				var_process := 5;
			END_IF
		5:
			gvl_elecylinder.fbi_gm_axisTransport.in_flg_run := FALSE;
			gvl_elecylinder.fbi_gm_axisPickUp.in_flg_run := FALSE;
			gvl_solv.fbi_gm_pickup.in_flg_run := FALSE;
			gvl_solv.fbi_gm_rotary.in_flg_run := FALSE;
			var_process := 6;
		6:
			trn_transportDone := TRUE;
		    
	END_CASE
END_IF
END_ACTION

ACTION waittingLens_active:
IF waittingLens._x AND waittingLens.x = FALSE THEN
	trn_waittingLensDone := FALSE;
ELSIF waittingLens._x AND waittingLens.x THEN
	IF gvl_gm.flg_requestPickup THEN
		trn_waittingLensDone := TRUE;
	END_IF
END_IF
END_ACTION

END_FUNCTION_BLOCK

// ---- FBs/fb_debuger.TcPOU
FUNCTION_BLOCK fb_debuger
VAR_INPUT
	in_flg_run: BOOL;
	in_flg_start: BOOL;
	in_var_cavQty: INT;
END_VAR
VAR_OUTPUT
	out_flg_gateLengthISSuccessed: BOOL;
	out_flg_dummySignal: BOOL;
	out_flg_lensSetDone: BOOL;
	out_flg_fiberSens: BOOL;
	out_flg_busy: BOOL;
	out_cav: INT;
END_VAR
VAR
	var_process: INT;
	var_cav: INT;
	delayTimer: TON;
END_VAR

IF in_flg_start AND in_flg_run THEN
	out_flg_busy := TRUE;
ELSE
	out_flg_busy := FALSE;
	var_process := 0;
	var_cav := gvl_param.var_productInfo[gvl_param.var_currentProductID].startCav - 1;
END_IF

CASE var_process OF
	0:
		out_flg_gateLengthISSuccessed := FALSE;
		out_flg_dummySignal := FALSE;
		out_flg_lensSetDone := FALSE;
		out_flg_fiberSens := FALSE;
		gvl_debug.cavConecctSkip := FALSE;
		delayTimer.IN := FALSE;
		IF out_flg_busy AND gvl_io.flg_requestLens THEN
			var_process := 1;
		END_IF
	1:
		gvl_debug.cavConecctSkip := TRUE;
		var_process := 2;
	2:
		//gate
		out_flg_gateLengthISSuccessed := TRUE;
		var_process := 3;
		
	3:
		//dummy signal
		IF gvl_debug.dummySignal THEN
			out_flg_dummySignal := TRUE;
			var_process := 4;
		ELSE
			var_process := 4;
		END_IF
	4:
		IF var_cav >= in_var_cavQty THEN
			var_cav := 1;
			out_cav := var_cav;
			var_process := 5;
		ELSE
			var_cav := var_cav + 1;
			out_cav := var_cav;
			var_process := 5;
		END_IF
	
	5:
		//lens set done
		delayTimer.IN := TRUE;
		out_flg_fiberSens := TRUE;
		IF delayTimer.Q THEN
			IF gvl_debug.flg_debug_run THEN
				out_flg_lensSetDone := TRUE;
				var_process := 0;
			END_IF
		END_IF
END_CASE
delayTimer(IN:= , PT:= T#3S , Q=> , ET=> );

END_FUNCTION_BLOCK

// ---- FBs/fb_gateLengthList.TcPOU
FUNCTION_BLOCK fb_gateLengthList
VAR_INPUT
END_VAR
VAR_OUTPUT
END_VAR
VAR
	fbi_R_TRIG: R_TRIG;
	flg_buf_gateLengthData: LREAL;
	var_process: INT;
	var_i: INT;
END_VAR

IF gvl_gm.var_buf_measurementCav <> 0 THEN
	fbi_R_TRIG(CLK:= gvl_auto.flg_gateData_Tx, Q=> );
END_IF


CASE var_process OF
	0:
		IF fbi_R_TRIG.Q THEN
			flg_buf_gateLengthData := DINT_TO_LREAL(gvl_io.var_gateLength)/10000;
			IF gvl_io.var_gateLength > gvl_param.var_productInfo[gvl_param.var_currentProductID].gateLength_max OR gvl_io.var_gateLength < gvl_param.var_productInfo[gvl_param.var_currentProductID].gateLength_min THEN
				flg_buf_gateLengthData := flg_buf_gateLengthData * -1;
			END_IF
			IF gvl_io.flg_gm_fiberSens THEN
				var_process := 10;
			END_IF
		END_IF
	10:
		FOR var_i := 49 TO 1 BY -1 DO
			IF gvl_visu.flg_btn_usingMeasurementSystem THEN
				gvl_visu.var_gateLengthList[var_i] := gvl_visu.var_gateLengthList[var_i - 1];
				gvl_visu.var_gateLengthListCav[gvl_gm.var_buf_measurementCav][var_i] := gvl_visu.var_gateLengthListCav[gvl_gm.var_buf_measurementCav][var_i - 1];
				IF var_i = 1 THEN
					gvl_visu.var_gateLengthList[0] := INT_TO_REAL(LREAL_TO_INT(flg_buf_gateLengthData*10000)/100)/100;
					gvl_visu.var_gateLengthListCav[gvl_gm.var_buf_measurementCav][0] := INT_TO_REAL(LREAL_TO_INT(flg_buf_gateLengthData*10000)/100)/100;		
					var_process := 0;
				END_IF
			ELSE
				gvl_visu.var_gateLengthList[var_i] := gvl_visu.var_gateLengthList[var_i - 1];
				gvl_visu.var_gateLengthListCav[gvl_auto.cavNo][var_i] := gvl_visu.var_gateLengthListCav[gvl_gm.var_buf_measurementCav][var_i - 1];
				IF var_i = 1 THEN
					gvl_visu.var_gateLengthList[0] := INT_TO_REAL(LREAL_TO_INT(flg_buf_gateLengthData*10000)/100)/100;
					gvl_visu.var_gateLengthListCav[gvl_auto.cavNo][0] := INT_TO_REAL(LREAL_TO_INT(flg_buf_gateLengthData*10000)/100)/100;			
					var_process := 0;
				END_IF
			END_IF
		END_FOR
	20:
		
END_CASE

END_FUNCTION_BLOCK

// ---- FBs/fb_dataSampling.TcPOU
FUNCTION_BLOCK fb_dataSampling
VAR_INPUT
	in_flg_run: BOOL;
	in_var_cavNo : INT;
	in_var_pocketNo : INT;
	in_var_gateLength : LREAL;
	in_var_date : DT;
	in_flg_nonDefective : BOOL;
	in_flg_defective : BOOL;
	in_flg_sample : BOOL;
	in_flg_reset : BOOL;
END_VAR
VAR_OUTPUT
END_VAR
VAR_IN_OUT
	ref_dataSet : s_DataSample;
END_VAR
VAR
	data : s_DataSample;

	fbi_r_trig: R_TRIG;
	fbi_reset: R_TRIG;
	var_i: INT;
	var_pocketNO: INT;
	var_cavNo: INT;

	fbi_setQty: R_TRIG;
END_VAR

fbi_r_trig(CLK:= in_flg_run, Q=> );
fbi_reset(CLK:= in_flg_reset, Q=> );

IF fbi_r_trig.Q THEN
	IF NOT in_flg_sample THEN
		IF in_flg_nonDefective AND NOT in_flg_defective THEN
			ref_dataSet.SetQty.cav[in_var_cavNo].nonDefectiveQty	:= ref_dataSet.SetQty.cav[in_var_cavNo].nonDefectiveQty + 1;
			FOR var_i := 500 TO 1 BY -1 DO
				ref_dataSet.DataSet[var_i].cav[in_var_cavNo].pocketNo[in_var_pocketNo].gateLength	:= ref_dataSet.DataSet[var_i - 1].cav[in_var_cavNo].pocketNo[in_var_pocketNo].gateLength;
				ref_dataSet.DataSet[var_i].cav[in_var_cavNo].pocketNo[in_var_pocketNo].setDate		:= ref_dataSet.DataSet[var_i - 1].cav[in_var_cavNo].pocketNo[in_var_pocketNo].setDate;
				IF var_i = 1 THEN
					ref_dataSet.DataSet[0].cav[in_var_cavNo].pocketNo[in_var_pocketNo].gateLength	:= in_var_gateLength;
					ref_dataSet.DataSet[0].cav[in_var_cavNo].pocketNo[in_var_pocketNo].setDate		:= DT_TO_STRING(in_var_date);
				END_IF
			END_FOR
		ELSIF NOT in_flg_nonDefective AND in_flg_defective THEN
			ref_dataSet.SetQty.cav[in_var_cavNo].defectiveQty		:= ref_dataSet.SetQty.cav[in_var_cavNo].defectiveQty + 1;
		END_IF
	END_IF
END_IF

IF fbi_reset.Q THEN
	FOR var_i := 0 TO 500 BY 1 DO
		FOR var_cavNo := 0 TO 8 BY 1 DO
			ref_dataSet.SetQty.cav[var_cavNo].nonDefectiveQty := 0;
			ref_dataSet.SetQty.cav[var_cavNo].defectiveQty := 0;
			FOR var_pocketNO := 0 TO 100 BY 1 DO
				ref_dataSet.DataSet[var_i].cav[in_var_cavNo].pocketNo[in_var_pocketNo].gateLength	:= 0;
				ref_dataSet.DataSet[var_i].cav[in_var_cavNo].pocketNo[in_var_pocketNo].setDate		:= '';
			END_FOR
		END_FOR
	END_FOR
END_IF

END_FUNCTION_BLOCK

// ---- FBs/gateMeasurementModule/fb_gm_removeLens.TcPOU
FUNCTION_BLOCK fb_gm_removeLens
VAR_INPUT
	in_flg_run: BOOL;
END_VAR
VAR_OUTPUT
	out_flg_Done: BOOL;
END_VAR
VAR
	SFCInit: BOOL;
	trn_checkVacDone: BOOL;
	trn_rmoveLensThetaDone: BOOL;
	var_process: INT;
	trn_removeLensDone: BOOL;
	trn_removeLen_stocker_eject_Done : BOOL;
	trn_removeLen_stocker_fiber_Done : BOOL;
	trn_removeLen_measurement_eject_Done : BOOL;
	trn_removeLen_measurement_fiber_Done : BOOL;
	timer: TON;
	timer2: TON;
END_VAR

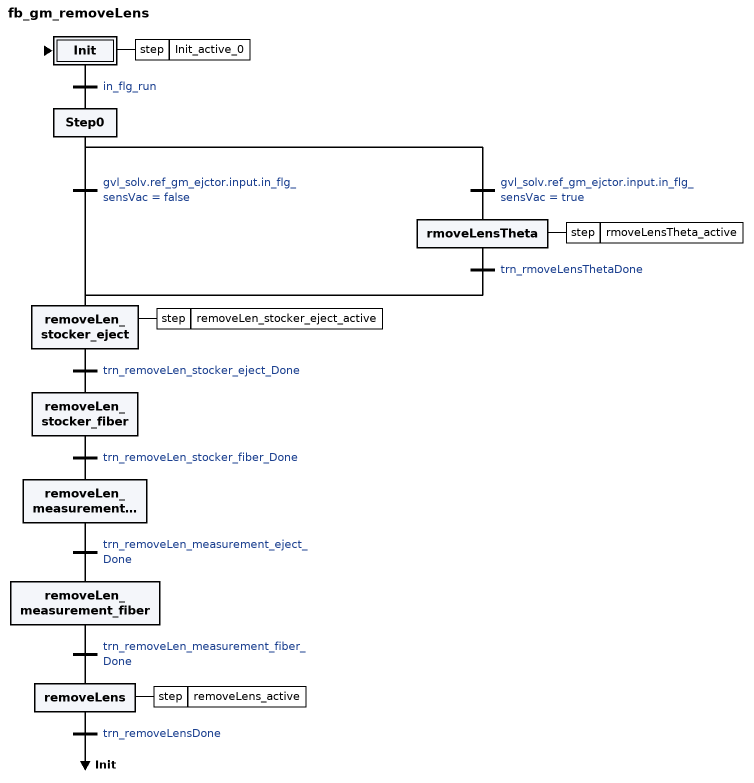
INITIAL_STEP Init:
    Init_active_0(N);  // step action
END_STEP
TRANSITION FROM Init TO Step0
    := in_flg_run;
END_TRANSITION
STEP Step0:
END_STEP
TRANSITION FROM Step0 TO removeLen_stocker_eject
    := gvl_solv.ref_gm_ejctor.input.in_flg_sensVac = false;
END_TRANSITION
TRANSITION FROM Step0 TO rmoveLensTheta
    := gvl_solv.ref_gm_ejctor.input.in_flg_sensVac = true;
END_TRANSITION
STEP rmoveLensTheta:
    rmoveLensTheta_active(N);  // step action
END_STEP
TRANSITION FROM rmoveLensTheta TO removeLen_stocker_eject
    := trn_rmoveLensThetaDone;
END_TRANSITION
STEP removeLen_stocker_eject:
    removeLen_stocker_eject_active(N);  // step action
END_STEP
TRANSITION FROM removeLen_stocker_eject TO removeLen_stocker_fiber
    := trn_removeLen_stocker_eject_Done;
END_TRANSITION
STEP removeLen_stocker_fiber:
END_STEP
TRANSITION FROM removeLen_stocker_fiber TO removeLen_measurement_eject
    := trn_removeLen_stocker_fiber_Done;
END_TRANSITION
STEP removeLen_measurement_eject:
END_STEP
TRANSITION FROM removeLen_measurement_eject TO removeLen_measurement_fiber
    := trn_removeLen_measurement_eject_Done;
END_TRANSITION
STEP removeLen_measurement_fiber:
END_STEP
TRANSITION FROM removeLen_measurement_fiber TO removeLens
    := trn_removeLen_measurement_fiber_Done;
END_TRANSITION
STEP removeLens:
    removeLens_active(N);  // step action
END_STEP
TRANSITION FROM removeLens TO Init
    := trn_removeLensDone;
END_TRANSITION

ACTION Init_active:
trn_removeLensDOne := false;
END_ACTION

ACTION Init_active_0:
out_flg_done := false;
END_ACTION

PROPERTY p_Init : BOOL
GET
p_Init := THIS^.SFCInit;
END_GET
SET
THIS^.SFCInit := p_Init;
END_SET
END_PROPERTY

ACTION removeLen_stocker_eject_active:
IF removeLen_stocker_eject._x AND removeLen_stocker_eject.x = FALSE THEN
	trn_removeLensDone := FALSE;
	timer.IN := FALSE;
	timer2.IN := FALSE;
	gvl_elecylinder.fbi_gm_axisPickUp.in_flg_run := FALSE;
	gvl_elecylinder.fbi_gm_axisPickUp.in_var_moveMode := eP_eleMoveMode.eleB;
	gvl_solv.fbi_gm_ejector.in_flg_run := FALSE;
	gvl_solv.fbi_gm_ejector.in_var_vacMode := eP_ejeVacMode.halt;
	gvl_axis.ref_r.Execute := FALSE;
	gvl_solv.fbi_gm_chuck.in_var_moveMode := eP_svMoveMode.svB;
	gvl_solv.fbi_gm_chuck.in_flg_run := FALSE;
	gvl_solv.fbi_gm_push.in_var_moveMode := eP_svMoveMode.svB;
	gvl_solv.fbi_gm_push.in_flg_run := FALSE;
	gvl_axis.ref_r.Position := gvl_param.var_productInfo[gvl_param.var_currentProductID].teachPos.gm_rotary.pickUp;
	var_process := 0;
ELSIF removeLen_stocker_eject._x AND removeLen_stocker_eject.x THEN
	CASE var_process OF
		0:
			IF gvl_io.flg_gm_fiberSens THEN
				var_process := 1;
			ELSE
				var_process := 100;
			END_IF
		1:
			
			
		
		
		100:
			trn_removeLensDone := TRUE;

	END_CASE
END_IF
END_ACTION

ACTION removeLens_active:
IF removeLens._x AND removeLens.x = FALSE THEN
	trn_removeLensDone := FALSE;
	timer.IN := FALSE;
	timer2.IN := FALSE;
	gvl_elecylinder.fbi_gm_axisPickUp.in_flg_run := FALSE;
	gvl_elecylinder.fbi_gm_axisPickUp.in_var_moveMode := eP_eleMoveMode.eleB;
	gvl_solv.fbi_gm_ejector.in_flg_run := FALSE;
	gvl_solv.fbi_gm_ejector.in_var_vacMode := eP_ejeVacMode.halt;
	gvl_axis.ref_r.Execute := FALSE;
	gvl_solv.fbi_gm_chuck.in_var_moveMode := eP_svMoveMode.svB;
	gvl_solv.fbi_gm_chuck.in_flg_run := FALSE;
	gvl_solv.fbi_gm_push.in_var_moveMode := eP_svMoveMode.svB;
	gvl_solv.fbi_gm_push.in_flg_run := FALSE;
	gvl_axis.ref_r.Position := gvl_param.var_productInfo[gvl_param.var_currentProductID].teachPos.gm_rotary.pickUp;
	var_process := 0;
ELSIF removeLens._x AND removeLens.x THEN
	CASE var_process OF
		0:
			IF gvl_io.flg_gm_fiberSens THEN
				//gvl_solv.fbi_gm_chuck.in_flg_run := TRUE;
				gvl_solv.fbi_gm_ejector.in_var_vacMode := eP_ejeVacMode.break;
				gvl_solv.fbi_gm_ejector.in_flg_run := TRUE;
				var_process := 15;
			ELSE
				gvl_solv.fbi_gm_ejector.in_var_vacMode := eP_ejeVacMode.break;
				gvl_solv.fbi_gm_ejector.in_flg_run := TRUE;
				var_process := 15;
			END_IF
		1:
			IF gvl_solv.fbi_gm_chuck.out_flg_Done THEN
				gvl_solv.fbi_gm_chuck.in_var_moveMode := eP_svMoveMode.svA;
				gvl_solv.fbi_gm_chuck.in_flg_run := FALSE;
				gvl_solv.fbi_gm_push.in_flg_run := TRUE;
				var_process := 2;
			END_IF
		2:
			IF gvl_solv.fbi_gm_push.out_flg_Done THEN
				gvl_solv.fbi_gm_push.in_var_moveMode := eP_svMoveMode.svA;
				gvl_solv.fbi_gm_push.in_flg_run := FALSE;
				var_process := 3;
			END_IF	
		3:
			gvl_axis.ref_r.Execute := TRUE;
			var_process := 4;
		4:
			IF gvl_axis.ref_r.Done THEN
				gvl_axis.ref_r.Execute := FALSE;
				var_process := 5;
			END_IF
		5:	
			gvl_solv.fbi_gm_ejector.in_flg_run := TRUE;
			gvl_elecylinder.fbi_gm_axisPickUp.in_flg_run := TRUE;
			var_process := 6;
		6:
			IF gvl_elecylinder.fbi_gm_axisPickUp.out_flg_Done THEN
				timer.IN := TRUE;
				gvl_elecylinder.fbi_gm_axisPickUp.in_flg_run := FALSE;
				var_process := 7;
			END_IF
		7:
			IF 	timer.Q THEN
				gvl_elecylinder.fbi_gm_axisPickUp.in_var_moveMode := eP_eleMoveMode.eleA;
				gvl_elecylinder.fbi_gm_axisPickUp.in_flg_run := FALSE;
				var_process := 8;
			END_IF
		8:
			gvl_solv.fbi_gm_chuck.in_flg_run := TRUE;
			gvl_solv.fbi_gm_push.in_flg_run := TRUE;
			var_process := 9;
		9:
			timer2.IN := TRUE;
			IF timer2.Q THEN
				var_process := 10;
			END_IF
			
		10:
			gvl_elecylinder.fbi_gm_axisPickUp.in_flg_run := TRUE;
			gvl_axis.ref_r.Position := gvl_param.var_productInfo[gvl_param.var_currentProductID].teachPos.gm_rotary.remove;
			var_process := 11;
		11:
			IF gvl_elecylinder.fbi_gm_axisPickUp.out_flg_Done THEN
				gvl_axis.ref_r.Execute := TRUE;
				gvl_solv.fbi_gm_ejector.in_flg_run := FALSE;
				gvl_solv.fbi_gm_ejector.in_var_vacMode := eP_ejeVacMode.break;
				var_process := 12;
			END_IF
		12:
			IF gvl_axis.ref_r.Done THEN
				gvl_axis.ref_r.Execute := FALSE;
				gvl_solv.fbi_gm_ejector.in_flg_run := TRUE;
				var_process := 13;
			END_IF
		13:
			IF gvl_solv.fbi_gm_ejector.out_flg_Done THEN
				gvl_axis.ref_r.Position := gvl_param.var_productInfo[gvl_param.var_currentProductID].teachPos.gm_rotary.origin;
				gvl_axis.ref_r.Execute := TRUE;
				var_process := 14;
			END_IF
		14:
			IF gvl_axis.ref_r.Done THEN
				gvl_axis.ref_r.Execute := FALSE;
				var_process := 15;
			END_IF
		15:
			gvl_solv.fbi_gm_ejector.in_flg_run := FALSE;
			out_flg_Done := TRUE;
			trn_removeLensDone := TRUE;
			
			
			
	END_CASE
timer(IN:= , PT:=T#0.5S , Q=> , ET=> );
timer2(IN:= , PT:=T#0.2S , Q=> , ET=> );
END_IF
END_ACTION

ACTION rmoveLensTheta_active:
IF rmoveLensTheta._x AND rmoveLensTheta.x = FALSE THEN
	var_process := 0;
	trn_rmoveLensThetaDone := FALSE;
	gvl_axis.ref_r.Execute := FALSE;
	gvl_solv.fbi_gm_ejector.in_flg_run := FALSE;
	gvl_solv.fbi_gm_ejector.in_var_vacMode := eP_ejeVacMode.break;
	gvl_axis.ref_r.Position := gvl_param.var_productInfo[gvl_param.var_currentProductID].teachPos.gm_rotary.remove;
ELSIF rmoveLensTheta._x AND rmoveLensTheta.x THEN
	CASE var_process OF
		0:
			gvl_axis.ref_r.Execute := TRUE;
			var_process := 1;
		1:
			IF gvl_axis.ref_r.Done THEN
				gvl_solv.fbi_gm_ejector.in_flg_run := TRUE;
				var_process := 2;
			END_IF
		2:
			IF gvl_solv.fbi_gm_ejector.out_flg_Done THEN
				var_process := 3;
			END_IF
		3:	
			gvl_axis.ref_r.Position := gvl_param.var_productInfo[gvl_param.var_currentProductID].teachPos.gm_rotary.pickUp;
			gvl_axis.ref_r.Execute := FALSE;
			var_process := 4;
		4:
			gvl_axis.ref_r.Execute := TRUE;
			var_process := 5;
		5:
			IF gvl_axis.ref_r.Done THEN
				trn_rmoveLensThetaDone := TRUE;
			END_IF
	END_CASE
END_IF
END_ACTION

END_FUNCTION_BLOCK

// ---- FBs/fb_motorController.TcPOU
FUNCTION_BLOCK fb_motorController
VAR_INPUT
	in_flg_run : BOOL;
END_VAR
VAR_OUTPUT
	out_flg_run : bool;
END_VAR
VAR
	flg_mototPowerRun: BOOL;
	flg_motorPowerReset: bool;
	fbi_delayTimerY: TON;
	fbi_delayTimerZ: TON;
	flg_rotaryPowerRun: BOOL;
	fbi_delayTimer1: TON;
END_VAR
VAR // added by the converter: edge detectors and wires of the graphical bodies
    _rt1, _rt2, _rt3, _rt4, _rt5, _rt6 : R_TRIG;
    _ft1, _ft2 : F_TRIG;
END_VAR

motorPower();
motorMoveAbs();
gm_rotary();
IF  gvl_param.var_currentMode = eP_programMode.manual OR gvl_param.var_currentMode = eP_programMode.error THEN
	motorJog();
END_IF
IF gvl_axis.axisX.NcToPlc.ActTorque > 500 THEN
	gvl_error.flg_axisXTorqueOver := TRUE;
ELSIF gvl_axis.axisY.NcToPlc.ActTorque > 500 THEN
	gvl_error.flg_axisYTorqueOver := TRUE;
ELSIF gvl_axis.axisZ.NcToPlc.ActTorque > 500 THEN
	gvl_error.flg_axisZTorqueOver := TRUE;
ELSIF gvl_axis.axisR.NcToPlc.ActTorque > 500 THEN
	gvl_error.flg_axisRTorqueOver := TRUE;
ELSE
	gvl_error.flg_axisXTorqueOver := FALSE;
	gvl_error.flg_axisYTorqueOver := FALSE;
	gvl_error.flg_axisZTorqueOver := FALSE;
	gvl_error.flg_axisRTorqueOver := FALSE;
END_IF

ACTION gm_rotary:
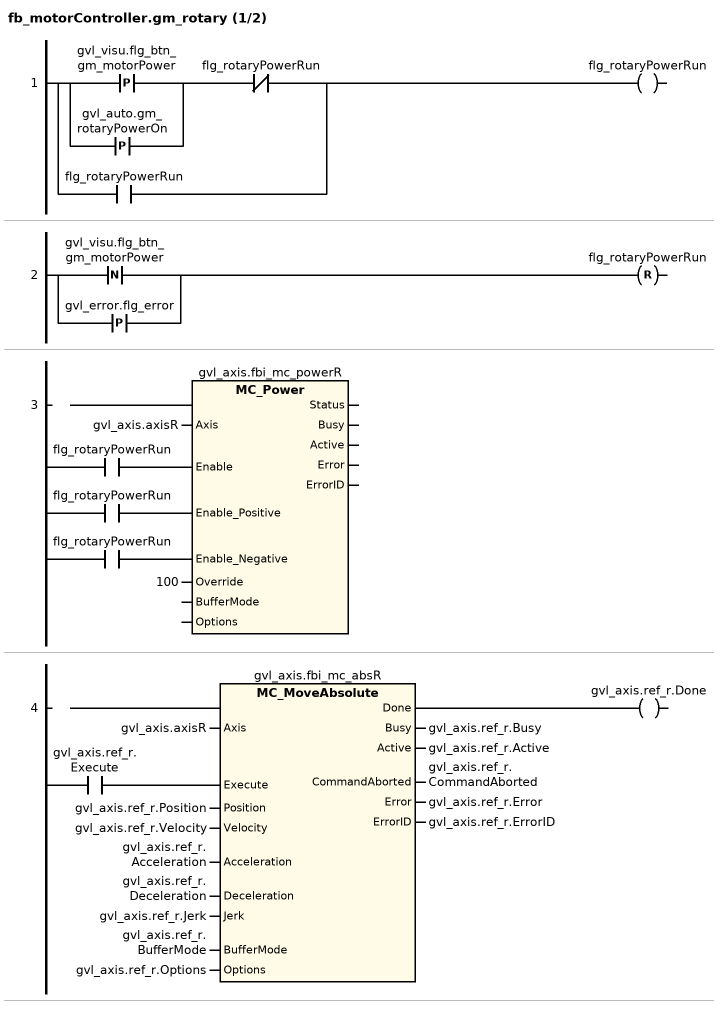
// NETWORK 1
_rt1(CLK := gvl_visu.flg_btn_gm_motorPower);
_rt2(CLK := gvl_auto.gm_rotaryPowerOn);
flg_rotaryPowerRun := (_rt1.Q OR _rt2.Q) AND NOT flg_rotaryPowerRun OR flg_rotaryPowerRun;

// NETWORK 2
_ft1(CLK := gvl_visu.flg_btn_gm_motorPower);
_rt3(CLK := gvl_error.flg_error);
flg_rotaryPowerRun R= _ft1.Q OR _rt3.Q;

// NETWORK 3
gvl_axis.fbi_mc_powerR(
    Axis := gvl_axis.axisR,
    Enable := flg_rotaryPowerRun,
    Enable_Positive := flg_rotaryPowerRun,
    Enable_Negative := flg_rotaryPowerRun,
    Override := 100); // MC_Power

